LIN {X 0.154,Y -380.012,Z 1004.456,A 0.000,B 0.000,C 90.000,E1 82.129} C_DIS
LIN {X 0.169,Y -370.321,Z 1004.447,A 0.000,B 0.000,C 90.000,E1 80.387} C_DIS
LIN {X 0.082,Y -360.354,Z 1004.437,A 0.000,B 0.000,C 90.000,E1 78.634} C_DIS
LIN {X 0.041,Y -345.465,Z 1004.422,A 0.000,B 0.000,C 90.000,E1 75.936} C_DIS
LIN {X -0.138,Y -331.066,Z 1004.406,A 0.000,B 0.000,C 90.000,E1 73.196} C_DIS
LIN {X -0.138,Y -318.755,Z 1004.393,A 0.000,B 0.000,C 90.000,E1 70.678} C_DIS
LIN {X -0.044,Y -308.159,Z 1004.380,A 0.000,B 0.000,C 90.000,E1 68.411} C_DIS
LIN {X -0.184,Y -294.870,Z 1004.364,A 0.000,B 0.000,C 90.000,E1 65.485} C_DIS
LIN {X -0.128,Y -284.811,Z 1004.351,A 0.000,B 0.000,C 90.000,E1 63.127} C_DIS
LIN {X -0.028,Y -274.834,Z 1004.337,A 0.000,B 0.000,C 90.000,E1 60.717} C_DIS
LIN {X -0.023,Y -264.962,Z 1004.324,A 0.000,B 0.000,C 90.000,E1 58.280} C_DIS
LIN {X 0.089,Y -252.725,Z 1004.306,A 0.000,B 0.000,C 90.000,E1 55.055} C_DIS
LIN {X -0.103,Y -242.379,Z 1004.290,A 0.000,B 0.000,C 90.000,E1 52.190} C_DIS
LIN {X -0.123,Y -231.354,Z 1004.271,A 0.000,B 0.000,C 90.000,E1 48.852} C_DIS
LIN {X -0.097,Y -222.061,Z 1004.254,A 0.000,B 0.000,C 90.000,E1 45.810} C_DIS
LIN {X 0.061,Y -212.191,Z 1004.235,A 0.000,B 0.000,C 90.000,E1 42.285} C_DIS
LIN {X 0.119,Y -203.993,Z 1004.217,A 0.000,B 0.000,C 90.000,E1 39.116} C_DIS
LIN {X 0.034,Y -196.376,Z 1004.200,A 0.000,B 0.000,C 90.000,E1 35.931} C_DIS
LIN {X 0.017,Y -189.584,Z 1004.182,A 0.000,B 0.000,C 90.000,E1 32.673} C_DIS
LIN {X 0.019,Y -183.573,Z 1004.163,A 0.000,B 0.000,C 90.000,E1 29.361} C_DIS
LIN {X -0.052,Y -178.371,Z 1004.145,A 0.000,B 0.000,C 90.000,E1 26.027} C_DIS
LIN {X -0.084,Y -173.934,Z 1004.126,A 0.000,B 0.000,C 90.000,E1 22.642} C_DIS
LIN {X -0.091,Y -170.157,Z 1004.107,A 0.000,B 0.000,C 90.000,E1 19.214} C_DIS
LIN {X 0.076,Y -166.471,Z 1004.083,A 0.000,B 0.000,C 90.000,E1 14.828} C_DIS
LIN {X -0.002,Y -163.812,Z 1004.058,A 0.000,B 0.000,C 90.000,E1 10.489} C_DIS
LIN {X 0.043,Y -161.757,Z 1004.019,A 0.000,B 0.000,C 90.000,E1 3.440} C_DIS
LIN {X 0.074,Y -163.118,Z 1003.963,A 0.000,B 0.000,C 90.000,E1 353.337} C_DIS
LIN {X -0.025,Y -165.817,Z 1003.934,A 0.000,B 0.000,C 90.000,E1 348.105} C_DIS
LIN {X -0.007,Y -169.285,Z 1003.910,A 0.000,B 0.000,C 90.000,E1 343.740} C_DIS
LIN {X -0.058,Y -172.872,Z 1003.890,A 0.000,B 0.000,C 90.000,E1 340.296} C_DIS
LIN {X -0.003,Y -177.301,Z 1003.871,A 0.000,B 0.000,C 90.000,E1 336.847} C_DIS
LIN {X -0.031,Y -182.552,Z 1003.852,A 0.000,B 0.000,C 90.000,E1 333.461} C_DIS
LIN {X 0.066,Y -188.584,Z 1003.834,A 0.000,B 0.000,C 90.000,E1 330.078} C_DIS
LIN {X 0.013,Y -195.305,Z 1003.815,A 0.000,B 0.000,C 90.000,E1 326.786} C_DIS
LIN {X -0.035,Y -202.588,Z 1003.797,A 0.000,B 0.000,C 90.000,E1 323.543} C_DIS
LIN {X 0.095,Y -211.472,Z 1003.777,A 0.000,B 0.000,C 90.000,E1 319.908} C_DIS
LIN {X 0.122,Y -220.912,Z 1003.758,A 0.000,B 0.000,C 90.000,E1 316.377} C_DIS
LIN {X 0.094,Y -231.213,Z 1003.739,A 0.000,B 0.000,C 90.000,E1 312.933} C_DIS
LIN {X 0.048,Y -236.546,Z 1003.730,A 0.000,B 0.000,C 90.000,E1 311.434} C_DIS
LIN {X 0.068,Y -244.132,Z 1003.720,A 0.000,B 0.000,C 90.000,E1 309.564} C_DIS
LIN {X 0.061,Y -252.554,Z 1003.710,A 0.000,B 0.000,C 90.000,E1 307.729} C_DIS
LIN {X -0.082,Y -263.737,Z 1003.698,A 0.000,B 0.000,C 90.000,E1 305.598} C_DIS
LIN {X 0.083,Y -280.210,Z 1003.682,A 0.000,B 0.000,C 90.000,E1 302.752} C_DIS
LIN {X -0.015,Y -295.611,Z 1003.669,A 0.000,B 0.000,C 90.000,E1 300.384} C_DIS
LIN {X 0.092,Y -314.496,Z 1003.654,A 0.000,B 0.000,C 90.000,E1 297.719} C_DIS
LIN {X -0.130,Y -330.163,Z 1003.643,A 0.000,B 0.000,C 90.000,E1 295.848} C_DIS
LIN {X 0.087,Y -352.097,Z 1003.630,A 0.000,B 0.000,C 90.000,E1 293.462} C_DIS
LIN {X -0.028,Y -374.171,Z 1003.619,A 0.000,B 0.000,C 90.000,E1 291.354} C_DIS
LIN {X -0.007,Y -390.076,Z 1003.610,A 0.000,B 0.000,C 90.000,E1 289.885} C_DIS
LIN {X -0.151,Y -400.861,Z 1003.605,A 0.000,B 0.000,C 90.000,E1 288.906} C_DIS
LIN {X 0.103,Y -411.395,Z 1003.599,A 0.000,B 0.000,C 90.000,E1 287.873} C_DIS
LIN {X 0.172,Y -418.988,Z 1003.595,A 0.000,B 0.000,C 90.000,E1 287.094} C_DIS
LIN {X 0.026,Y -428.704,Z 1003.589,A 0.000,B 0.000,C 90.000,E1 286.079} C_DIS
LIN {X -0.072,Y -435.798,Z 1003.585,A 0.000,B 0.000,C 90.000,E1 285.300} C_DIS
LIN {X -0.131,Y -444.841,Z 1003.579,A 0.000,B 0.000,C 90.000,E1 284.245} C_DIS
LIN {X 0.030,Y -453.358,Z 1003.573,A 0.000,B 0.000,C 90.000,E1 283.175} C_DIS
LIN {X 0.188,Y -461.140,Z 1003.567,A 0.000,B 0.000,C 90.000,E1 282.119} C_DIS
LIN {X -0.108,Y -468.076,Z 1003.562,A 0.000,B 0.000,C 90.000,E1 281.130} C_DIS
LIN {X -0.096,Y -472.803,Z 1003.558,A 0.000,B 0.000,C 90.000,E1 280.366} C_DIS
LIN {X -0.133,Y -476.901,Z 1003.553,A 0.000,B 0.000,C 90.000,E1 279.613} C_DIS
LIN {X -0.128,Y -480.362,Z 1003.549,A 0.000,B 0.000,C 90.000,E1 278.859} C_DIS
LIN {X -0.094,Y -483.236,Z 1003.545,A 0.000,B 0.000,C 90.000,E1 278.106} C_DIS
LIN {X 0.077,Y -484.811,Z 1003.542,A 0.000,B 0.000,C 90.000,E1 277.587} C_DIS
LIN {X -0.222,Y -486.171,Z 1003.539,A 0.000,B 0.000,C 90.000,E1 277.125} C_DIS
LIN {X 0.173,Y -488.167,Z 1003.534,A 0.000,B 0.000,C 90.000,E1 276.087} C_DIS
LIN {X -0.104,Y -488.752,Z 1003.531,A 0.000,B 0.000,C 90.000,E1 275.625} C_DIS
LIN {X 0.108,Y -489.034,Z 1003.528,A 0.000,B 0.000,C 90.000,E1 275.106} C_DIS
LIN {X -0.166,Y -488.846,Z 1003.526,A 0.000,B 0.000,C 90.000,E1 274.645} C_DIS
LIN {X 0.012,Y -488.231,Z 1003.523,A 0.000,B 0.000,C 90.000,E1 274.131} C_DIS
LIN {X 0.224,Y -487.021,Z 1003.520,A 0.000,B 0.000,C 90.000,E1 273.612} C_DIS
LIN {X -0.084,Y -485.248,Z 1003.517,A 0.000,B 0.000,C 90.000,E1 273.154} C_DIS
LIN {X 0.113,Y -482.887,Z 1003.515,A 0.000,B 0.000,C 90.000,E1 272.636} C_DIS
LIN {X -0.211,Y -479.755,Z 1003.512,A 0.000,B 0.000,C 90.000,E1 272.178} C_DIS
LIN {X -0.054,Y -475.746,Z 1003.509,A 0.000,B 0.000,C 90.000,E1 271.661} C_DIS
LIN {X 0.065,Y -470.779,Z 1003.506,A 0.000,B 0.000,C 90.000,E1 271.146} C_DIS
LIN {X -0.119,Y -464.970,Z 1003.504,A 0.000,B 0.000,C 90.000,E1 270.688} C_DIS
LIN {X 0.155,Y -458.759,Z 1003.501,A 0.000,B 0.000,C 90.000,E1 270.229} C_DIS
LIN {X -0.051,Y -451.942,Z 1003.499,A 0.000,B 0.000,C 90.000,E1 269.885} C_DIS
LIN {X -0.182,Y -444.964,Z 1003.498,A 0.000,B 0.000,C 90.000,E1 269.599} C_DIS
LIN {X 0.077,Y -437.435,Z 1003.496,A 0.000,B 0.000,C 90.000,E1 269.312} C_DIS
LIN {X -0.119,Y -429.221,Z 1003.495,A 0.000,B 0.000,C 90.000,E1 269.141} C_DIS
LIN {X 0.095,Y -420.520,Z 1003.494,A 0.000,B 0.000,C 90.000,E1 268.969} C_DIS
LIN {X -0.086,Y -406.679,Z 1003.494,A 0.000,B 0.000,C 90.000,E1 268.854} C_DIS
LIN {X 0.121,Y -400.216,Z 1003.493,A 0.000,B 0.000,C 90.000,E1 268.797} C_DIS
LIN {X 0.026,Y -181.275,Z 1003.493,A 0.000,B 0.000,C 90.000,E1 268.797} C_DIS
LIN {X 0.089,Y -180.880,Z 1003.473,A 0.000,B 0.000,C 90.000,E1 265.065} C_DIS
LIN {X -0.032,Y -178.999,Z 1003.445,A 0.000,B 0.000,C 90.000,E1 260.038} C_DIS
LIN {X 0.062,Y -178.594,Z 1003.440,A 0.000,B 0.000,C 90.000,E1 259.162} C_DIS
LIN {X -0.044,Y -175.646,Z 1003.412,A 0.000,B 0.000,C 90.000,E1 254.102} C_DIS
LIN {X -0.039,Y -172.365,Z 1003.388,A 0.000,B 0.000,C 90.000,E1 249.826} C_DIS
LIN {X -0.024,Y -171.154,Z 1003.378,A 0.000,B 0.000,C 90.000,E1 248.103} C_DIS
LIN {X 0.020,Y -167.455,Z 1003.354,A 0.000,B 0.000,C 90.000,E1 243.768} C_DIS
LIN {X -0.046,Y -166.852,Z 1003.349,A 0.000,B 0.000,C 90.000,E1 242.922} C_DIS
LIN {X 0.018,Y -162.836,Z 1003.325,A 0.000,B 0.000,C 90.000,E1 238.535} C_DIS
LIN {X -0.007,Y -161.520,Z 1003.315,A 0.000,B 0.000,C 90.000,E1 236.786} C_DIS
LIN {X 0.034,Y -157.519,Z 1003.291,A 0.000,B 0.000,C 90.000,E1 232.351} C_DIS
LIN {X -0.033,Y -155.543,Z 1003.276,A 0.000,B 0.000,C 90.000,E1 229.703} C_DIS
LIN {X 0.009,Y -151.837,Z 1003.251,A 0.000,B 0.000,C 90.000,E1 225.202} C_DIS
LIN {X -0.083,Y -150.054,Z 1003.236,A 0.000,B 0.000,C 90.000,E1 222.528} C_DIS
LIN {X 0.042,Y -146.866,Z 1003.211,A 0.000,B 0.000,C 90.000,E1 217.935} C_DIS
LIN {X -0.060,Y -145.451,Z 1003.196,A 0.000,B 0.000,C 90.000,E1 215.231} C_DIS
LIN {X 0.054,Y -142.868,Z 1003.170,A 0.000,B 0.000,C 90.000,E1 210.590} C_DIS
LIN {X -0.020,Y -141.485,Z 1003.150,A 0.000,B 0.000,C 90.000,E1 206.924} C_DIS
LIN {X -0.034,Y -139.383,Z 1003.113,A 0.000,B 0.000,C 90.000,E1 200.429} C_DIS
LIN {X -0.046,Y -138.838,Z 1003.098,A 0.000,B 0.000,C 90.000,E1 197.638} C_DIS
LIN {X 0.015,Y -138.354,Z 1003.056,A 0.000,B 0.000,C 90.000,E1 190.141} C_DIS
LIN {X 0.010,Y -139.522,Z 1003.004,A 0.000,B 0.000,C 90.000,E1 180.802} C_DIS
LIN {X -0.050,Y -141.187,Z 1002.973,A 0.000,B 0.000,C 90.000,E1 175.241} C_DIS
LIN {X 0.063,Y -142.564,Z 1002.958,A 0.000,B 0.000,C 90.000,E1 172.413} C_DIS
LIN {X 0.018,Y -144.848,Z 1002.932,A 0.000,B 0.000,C 90.000,E1 167.813} C_DIS
LIN {X -0.027,Y -147.473,Z 1002.912,A 0.000,B 0.000,C 90.000,E1 164.157} C_DIS
LIN {X -0.001,Y -150.058,Z 1002.892,A 0.000,B 0.000,C 90.000,E1 160.496} C_DIS
LIN {X 0.004,Y -153.403,Z 1002.872,A 0.000,B 0.000,C 90.000,E1 156.869} C_DIS
LIN {X 0.051,Y -155.934,Z 1002.857,A 0.000,B 0.000,C 90.000,E1 154.152} C_DIS
LIN {X 0.024,Y -159.802,Z 1002.837,A 0.000,B 0.000,C 90.000,E1 150.589} C_DIS
LIN {X 0.010,Y -162.042,Z 1002.827,A 0.000,B 0.000,C 90.000,E1 148.820} C_DIS
LIN {X -0.016,Y -166.238,Z 1002.807,A 0.000,B 0.000,C 90.000,E1 145.308} C_DIS
LIN {X -0.015,Y -171.255,Z 1002.788,A 0.000,B 0.000,C 90.000,E1 141.823} C_DIS
LIN {X -0.093,Y -176.144,Z 1002.769,A 0.000,B 0.000,C 90.000,E1 138.405} C_DIS
LIN {X 0.023,Y -180.413,Z 1002.755,A 0.000,B 0.000,C 90.000,E1 135.810} C_DIS
LIN {X -0.001,Y -185.819,Z 1002.736,A 0.000,B 0.000,C 90.000,E1 132.447} C_DIS
LIN {X 0.053,Y -190.439,Z 1002.722,A 0.000,B 0.000,C 90.000,E1 129.930} C_DIS
LIN {X -0.111,Y -196.231,Z 1002.703,A 0.000,B 0.000,C 90.000,E1 126.664} C_DIS
LIN {X -0.025,Y -300.780,Z 1002.703,A 0.000,B 0.000,C 90.000,E1 126.629} C_DIS
LIN {X 0.004,Y -302.851,Z 1002.703,A 0.000,B 0.000,C 90.000,E1 126.583} C_DIS
LIN {X 0.105,Y -306.723,Z 1002.702,A 0.000,B 0.000,C 90.000,E1 126.377} C_DIS
LIN {X -0.041,Y -309.025,Z 1002.701,A 0.000,B 0.000,C 90.000,E1 126.217} C_DIS
LIN {X 0.165,Y -312.203,Z 1002.699,A 0.000,B 0.000,C 90.000,E1 125.804} C_DIS
LIN {X -0.006,Y -314.146,Z 1002.697,A 0.000,B 0.000,C 90.000,E1 125.518} C_DIS
LIN {X 0.080,Y -315.663,Z 1002.696,A 0.000,B 0.000,C 90.000,E1 125.185} C_DIS
LIN {X 0.120,Y -317.903,Z 1002.692,A 0.000,B 0.000,C 90.000,E1 124.532} C_DIS
LIN {X -0.113,Y -328.902,Z 1002.674,A 0.000,B 0.000,C 90.000,E1 121.386} C_DIS
LIN {X -0.080,Y -340.185,Z 1002.659,A 0.000,B 0.000,C 90.000,E1 118.565} C_DIS
LIN {X -0.035,Y -352.884,Z 1002.643,A 0.000,B 0.000,C 90.000,E1 115.796} C_DIS
LIN {X 0.074,Y -367.106,Z 1002.628,A 0.000,B 0.000,C 90.000,E1 113.078} C_DIS
LIN {X 0.030,Y -381.133,Z 1002.615,A 0.000,B 0.000,C 90.000,E1 110.737} C_DIS
LIN {X 0.205,Y -396.566,Z 1002.602,A 0.000,B 0.000,C 90.000,E1 108.417} C_DIS
LIN {X 0.011,Y -413.514,Z 1002.590,A 0.000,B 0.000,C 90.000,E1 106.205} C_DIS
LIN {X 0.123,Y -432.099,Z 1002.578,A 0.000,B 0.000,C 90.000,E1 104.008} C_DIS
LIN {X -0.022,Y -451.998,Z 1002.566,A 0.000,B 0.000,C 90.000,E1 101.951} C_DIS
LIN {X 0.102,Y -467.286,Z 1002.558,A 0.000,B 0.000,C 90.000,E1 100.489} C_DIS
LIN {X 0.122,Y -469.335,Z 1002.557,A 0.000,B 0.000,C 90.000,E1 100.254} C_DIS
LIN {X -0.030,Y -471.015,Z 1002.556,A 0.000,B 0.000,C 90.000,E1 100.018} C_DIS
LIN {X -0.183,Y -472.276,Z 1002.554,A 0.000,B 0.000,C 90.000,E1 99.782} C_DIS
LIN {X -0.082,Y -473.833,Z 1002.551,A 0.000,B 0.000,C 90.000,E1 99.265} C_DIS
LIN {X 0.030,Y -474.341,Z 1002.549,A 0.000,B 0.000,C 90.000,E1 98.746} C_DIS
LIN {X 0.223,Y -473.887,Z 1002.546,A 0.000,B 0.000,C 90.000,E1 98.219} C_DIS
LIN {X -0.121,Y -472.404,Z 1002.543,A 0.000,B 0.000,C 90.000,E1 97.757} C_DIS
LIN {X 0.145,Y -471.200,Z 1002.542,A 0.000,B 0.000,C 90.000,E1 97.473} C_DIS
LIN {X 0.112,Y -466.100,Z 1002.537,A 0.000,B 0.000,C 90.000,E1 96.720} C_DIS
LIN {X -0.140,Y -455.701,Z 1002.529,A 0.000,B 0.000,C 90.000,E1 95.220} C_DIS
LIN {X -0.105,Y -436.571,Z 1002.513,A 0.000,B 0.000,C 90.000,E1 92.350} C_DIS
LIN {X 0.100,Y -425.250,Z 1002.503,A 0.000,B 0.000,C 90.000,E1 90.458} C_DIS
LIN {X 0.013,Y -408.885,Z 1002.486,A 0.000,B 0.000,C 90.000,E1 87.478} C_DIS
LIN {X 0.033,Y -399.955,Z 1002.477,A 0.000,B 0.000,C 90.000,E1 85.812} C_DIS
LIN {X -0.051,Y -389.282,Z 1002.466,A 0.000,B 0.000,C 90.000,E1 83.856} C_DIS
LIN {X 0.037,Y -379.912,Z 1002.456,A 0.000,B 0.000,C 90.000,E1 82.129} C_DIS
LIN {X 0.054,Y -370.238,Z 1002.447,A 0.000,B 0.000,C 90.000,E1 80.387} C_DIS
LIN {X -0.032,Y -360.282,Z 1002.437,A 0.000,B 0.000,C 90.000,E1 78.634} C_DIS
LIN {X -0.070,Y -345.356,Z 1002.422,A 0.000,B 0.000,C 90.000,E1 75.936} C_DIS
LIN {X 0.068,Y -330.961,Z 1002.406,A 0.000,B 0.000,C 90.000,E1 73.142} C_DIS
LIN {X 0.160,Y -318.687,Z 1002.392,A 0.000,B 0.000,C 90.000,E1 70.604} C_DIS
LIN {X -0.151,Y -308.077,Z 1002.380,A 0.000,B 0.000,C 90.000,E1 68.411} C_DIS
LIN {X 0.104,Y -294.795,Z 1002.364,A 0.000,B 0.000,C 90.000,E1 65.409} C_DIS
LIN {X 0.025,Y -284.744,Z 1002.350,A 0.000,B 0.000,C 90.000,E1 63.076} C_DIS
LIN {X 0.112,Y -274.750,Z 1002.337,A 0.000,B 0.000,C 90.000,E1 60.667} C_DIS
LIN {X -0.061,Y -263.473,Z 1002.322,A 0.000,B 0.000,C 90.000,E1 57.916} C_DIS
LIN {X 0.016,Y -251.296,Z 1002.304,A 0.000,B 0.000,C 90.000,E1 54.689} C_DIS
LIN {X -0.020,Y -239.775,Z 1002.286,A 0.000,B 0.000,C 90.000,E1 51.412} C_DIS
LIN {X 0.025,Y -228.872,Z 1002.267,A 0.000,B 0.000,C 90.000,E1 48.038} C_DIS
LIN {X 0.050,Y -218.580,Z 1002.248,A 0.000,B 0.000,C 90.000,E1 44.595} C_DIS
LIN {X -0.069,Y -209.973,Z 1002.231,A 0.000,B 0.000,C 90.000,E1 41.515} C_DIS
LIN {X -0.033,Y -201.928,Z 1002.213,A 0.000,B 0.000,C 90.000,E1 38.338} C_DIS
LIN {X 0.002,Y -194.542,Z 1002.195,A 0.000,B 0.000,C 90.000,E1 35.105} C_DIS
LIN {X 0.101,Y -187.950,Z 1002.177,A 0.000,B 0.000,C 90.000,E1 31.799} C_DIS
LIN {X 0.061,Y -182.166,Z 1002.158,A 0.000,B 0.000,C 90.000,E1 28.487} C_DIS
LIN {X -0.051,Y -177.168,Z 1002.140,A 0.000,B 0.000,C 90.000,E1 25.155} C_DIS
LIN {X 0.053,Y -172.900,Z 1002.121,A 0.000,B 0.000,C 90.000,E1 21.716} C_DIS
LIN {X -0.039,Y -169.318,Z 1002.102,A 0.000,B 0.000,C 90.000,E1 18.308} C_DIS
LIN {X 0.013,Y -165.847,Z 1002.078,A 0.000,B 0.000,C 90.000,E1 13.953} C_DIS
LIN {X 0.054,Y -163.078,Z 1002.048,A 0.000,B 0.000,C 90.000,E1 8.690} C_DIS
LIN {X 0.006,Y -163.856,Z 1001.953,A 0.000,B 0.000,C 90.000,E1 351.602} C_DIS
LIN {X -0.017,Y -166.435,Z 1001.929,A 0.000,B 0.000,C 90.000,E1 347.229} C_DIS
LIN {X 0.057,Y -170.137,Z 1001.905,A 0.000,B 0.000,C 90.000,E1 342.851} C_DIS
LIN {X 0.079,Y -173.939,Z 1001.886,A 0.000,B 0.000,C 90.000,E1 339.390} C_DIS
LIN {X -0.009,Y -178.575,Z 1001.867,A 0.000,B 0.000,C 90.000,E1 335.997} C_DIS
LIN {X -0.018,Y -184.040,Z 1001.848,A 0.000,B 0.000,C 90.000,E1 332.615} C_DIS
LIN {X -0.047,Y -190.271,Z 1001.829,A 0.000,B 0.000,C 90.000,E1 329.282} C_DIS
LIN {X 0.044,Y -197.117,Z 1001.811,A 0.000,B 0.000,C 90.000,E1 325.960} C_DIS
LIN {X 0.041,Y -204.566,Z 1001.793,A 0.000,B 0.000,C 90.000,E1 322.718} C_DIS
LIN {X 0.032,Y -213.593,Z 1001.773,A 0.000,B 0.000,C 90.000,E1 319.138} C_DIS
LIN {X -0.043,Y -223.147,Z 1001.754,A 0.000,B 0.000,C 90.000,E1 315.648} C_DIS
LIN {X 0.101,Y -231.183,Z 1001.739,A 0.000,B 0.000,C 90.000,E1 312.933} C_DIS
LIN {X 0.055,Y -236.542,Z 1001.730,A 0.000,B 0.000,C 90.000,E1 311.434} C_DIS
LIN {X 0.066,Y -245.822,Z 1001.718,A 0.000,B 0.000,C 90.000,E1 309.197} C_DIS
LIN {X 0.081,Y -254.420,Z 1001.708,A 0.000,B 0.000,C 90.000,E1 307.363} C_DIS
LIN {X -0.125,Y -267.785,Z 1001.694,A 0.000,B 0.000,C 90.000,E1 304.898} C_DIS
LIN {X -0.006,Y -284.641,Z 1001.678,A 0.000,B 0.000,C 90.000,E1 302.084} C_DIS
LIN {X -0.140,Y -304.900,Z 1001.661,A 0.000,B 0.000,C 90.000,E1 299.077} C_DIS
LIN {X 0.075,Y -319.636,Z 1001.651,A 0.000,B 0.000,C 90.000,E1 297.078} C_DIS
LIN {X -0.039,Y -335.857,Z 1001.640,A 0.000,B 0.000,C 90.000,E1 295.207} C_DIS
LIN {X -0.083,Y -355.063,Z 1001.629,A 0.000,B 0.000,C 90.000,E1 293.206} C_DIS
LIN {X -0.172,Y -373.890,Z 1001.619,A 0.000,B 0.000,C 90.000,E1 291.408} C_DIS
LIN {X 0.029,Y -390.042,Z 1001.610,A 0.000,B 0.000,C 90.000,E1 289.885} C_DIS
LIN {X -0.120,Y -403.318,Z 1001.604,A 0.000,B 0.000,C 90.000,E1 288.671} C_DIS
LIN {X 0.193,Y -411.201,Z 1001.599,A 0.000,B 0.000,C 90.000,E1 287.873} C_DIS
LIN {X 0.238,Y -418.847,Z 1001.595,A 0.000,B 0.000,C 90.000,E1 287.094} C_DIS
LIN {X -0.109,Y -428.758,Z 1001.589,A 0.000,B 0.000,C 90.000,E1 286.079} C_DIS
LIN {X 0.123,Y -435.945,Z 1001.585,A 0.000,B 0.000,C 90.000,E1 285.245} C_DIS
LIN {X 0.073,Y -444.940,Z 1001.579,A 0.000,B 0.000,C 90.000,E1 284.189} C_DIS
LIN {X 0.240,Y -453.474,Z 1001.573,A 0.000,B 0.000,C 90.000,E1 283.119} C_DIS
LIN {X 0.133,Y -459.356,Z 1001.569,A 0.000,B 0.000,C 90.000,E1 282.355} C_DIS
LIN {X -0.184,Y -466.509,Z 1001.563,A 0.000,B 0.000,C 90.000,E1 281.366} C_DIS
LIN {X -0.189,Y -471.390,Z 1001.559,A 0.000,B 0.000,C 90.000,E1 280.602} C_DIS
LIN {X -0.234,Y -475.696,Z 1001.555,A 0.000,B 0.000,C 90.000,E1 279.849} C_DIS
LIN {X -0.167,Y -479.383,Z 1001.550,A 0.000,B 0.000,C 90.000,E1 279.086} C_DIS
LIN {X -0.020,Y -481.514,Z 1001.548,A 0.000,B 0.000,C 90.000,E1 278.568} C_DIS
LIN {X 0.144,Y -483.361,Z 1001.545,A 0.000,B 0.000,C 90.000,E1 278.049} C_DIS
LIN {X -0.164,Y -484.952,Z 1001.542,A 0.000,B 0.000,C 90.000,E1 277.587} C_DIS
LIN {X 0.020,Y -486.323,Z 1001.539,A 0.000,B 0.000,C 90.000,E1 277.068} C_DIS
LIN {X 0.215,Y -487.451,Z 1001.536,A 0.000,B 0.000,C 90.000,E1 276.549} C_DIS
LIN {X -0.067,Y -488.308,Z 1001.534,A 0.000,B 0.000,C 90.000,E1 276.087} C_DIS
LIN {X 0.143,Y -488.899,Z 1001.531,A 0.000,B 0.000,C 90.000,E1 275.568} C_DIS
LIN {X -0.131,Y -489.104,Z 1001.528,A 0.000,B 0.000,C 90.000,E1 275.106} C_DIS
LIN {X 0.084,Y -488.932,Z 1001.526,A 0.000,B 0.000,C 90.000,E1 274.588} C_DIS
LIN {X -0.225,Y -488.308,Z 1001.523,A 0.000,B 0.000,C 90.000,E1 274.131} C_DIS
LIN {X -0.012,Y -487.129,Z 1001.520,A 0.000,B 0.000,C 90.000,E1 273.612} C_DIS
LIN {X 0.193,Y -485.347,Z 1001.517,A 0.000,B 0.000,C 90.000,E1 273.094} C_DIS
LIN {X -0.120,Y -482.933,Z 1001.515,A 0.000,B 0.000,C 90.000,E1 272.636} C_DIS
LIN {X 0.038,Y -479.770,Z 1001.512,A 0.000,B 0.000,C 90.000,E1 272.121} C_DIS
LIN {X 0.193,Y -475.730,Z 1001.509,A 0.000,B 0.000,C 90.000,E1 271.604} C_DIS
LIN {X -0.161,Y -470.689,Z 1001.506,A 0.000,B 0.000,C 90.000,E1 271.146} C_DIS
LIN {X -0.233,Y -467.980,Z 1001.505,A 0.000,B 0.000,C 90.000,E1 270.917} C_DIS
LIN {X -0.157,Y -461.996,Z 1001.502,A 0.000,B 0.000,C 90.000,E1 270.458} C_DIS
LIN {X -0.087,Y -455.556,Z 1001.500,A 0.000,B 0.000,C 90.000,E1 270.057} C_DIS
LIN {X 0.006,Y -448.671,Z 1001.498,A 0.000,B 0.000,C 90.000,E1 269.714} C_DIS
LIN {X 0.090,Y -441.537,Z 1001.497,A 0.000,B 0.000,C 90.000,E1 269.427} C_DIS
LIN {X 0.141,Y -433.909,Z 1001.496,A 0.000,B 0.000,C 90.000,E1 269.198} C_DIS
LIN {X 0.159,Y -425.715,Z 1001.495,A 0.000,B 0.000,C 90.000,E1 269.026} C_DIS
LIN {X 0.096,Y -417.151,Z 1001.494,A 0.000,B 0.000,C 90.000,E1 268.912} C_DIS
LIN {X 0.117,Y -404.897,Z 1001.493,A 0.000,B 0.000,C 90.000,E1 268.797} C_DIS
LIN {X -0.025,Y -399.475,Z 1001.493,A 0.000,B 0.000,C 90.000,E1 268.797} C_DIS
LIN {X -0.032,Y -181.272,Z 1001.493,A 0.000,B 0.000,C 90.000,E1 268.797} C_DIS
LIN {X 0.048,Y -180.906,Z 1001.474,A 0.000,B 0.000,C 90.000,E1 265.355} C_DIS
LIN {X -0.059,Y -180.690,Z 1001.470,A 0.000,B 0.000,C 90.000,E1 264.546} C_DIS
LIN {X 0.019,Y -178.773,Z 1001.441,A 0.000,B 0.000,C 90.000,E1 259.454} C_DIS
LIN {X -0.078,Y -175.819,Z 1001.413,A 0.000,B 0.000,C 90.000,E1 254.393} C_DIS
LIN {X -0.076,Y -172.008,Z 1001.385,A 0.000,B 0.000,C 90.000,E1 249.263} C_DIS
LIN {X -0.100,Y -171.425,Z 1001.380,A 0.000,B 0.000,C 90.000,E1 248.411} C_DIS
LIN {X -0.044,Y -167.663,Z 1001.356,A 0.000,B 0.000,C 90.000,E1 244.076} C_DIS
LIN {X -0.104,Y -166.333,Z 1001.346,A 0.000,B 0.000,C 90.000,E1 242.359} C_DIS
LIN {X 0.029,Y -163.070,Z 1001.327,A 0.000,B 0.000,C 90.000,E1 238.820} C_DIS
LIN {X -0.059,Y -161.009,Z 1001.312,A 0.000,B 0.000,C 90.000,E1 236.215} C_DIS
LIN {X 0.051,Y -157.753,Z 1001.293,A 0.000,B 0.000,C 90.000,E1 232.637} C_DIS
LIN {X -0.011,Y -155.791,Z 1001.278,A 0.000,B 0.000,C 90.000,E1 229.989} C_DIS
LIN {X 0.044,Y -152.044,Z 1001.253,A 0.000,B 0.000,C 90.000,E1 225.486} C_DIS
LIN {X 0.062,Y -150.294,Z 1001.238,A 0.000,B 0.000,C 90.000,E1 222.771} C_DIS
LIN {X -0.013,Y -147.041,Z 1001.213,A 0.000,B 0.000,C 90.000,E1 218.257} C_DIS
LIN {X -0.021,Y -145.621,Z 1001.197,A 0.000,B 0.000,C 90.000,E1 215.518} C_DIS
LIN {X -0.021,Y -143.005,Z 1001.172,A 0.000,B 0.000,C 90.000,E1 210.924} C_DIS
LIN {X 0.036,Y -141.631,Z 1001.151,A 0.000,B 0.000,C 90.000,E1 207.206} C_DIS
LIN {X -0.039,Y -139.436,Z 1001.115,A 0.000,B 0.000,C 90.000,E1 200.737} C_DIS
LIN {X 0.015,Y -139.167,Z 1001.105,A 0.000,B 0.000,C 90.000,E1 198.852} C_DIS
LIN {X 0.048,Y -138.317,Z 1001.053,A 0.000,B 0.000,C 90.000,E1 189.500} C_DIS
LIN {X 0.059,Y -139.475,Z 1001.006,A 0.000,B 0.000,C 90.000,E1 181.088} C_DIS
LIN {X 0.001,Y -141.055,Z 1000.975,A 0.000,B 0.000,C 90.000,E1 175.527} C_DIS
LIN {X -0.045,Y -142.427,Z 1000.960,A 0.000,B 0.000,C 90.000,E1 172.761} C_DIS
LIN {X 0.016,Y -144.664,Z 1000.934,A 0.000,B 0.000,C 90.000,E1 168.117} C_DIS
LIN {X -0.001,Y -147.247,Z 1000.914,A 0.000,B 0.000,C 90.000,E1 164.448} C_DIS
LIN {X 0.017,Y -150.565,Z 1000.888,A 0.000,B 0.000,C 90.000,E1 159.880} C_DIS
LIN {X -0.044,Y -154.033,Z 1000.868,A 0.000,B 0.000,C 90.000,E1 156.282} C_DIS
LIN {X 0.024,Y -157.449,Z 1000.848,A 0.000,B 0.000,C 90.000,E1 152.666} C_DIS
LIN {X -0.027,Y -161.667,Z 1000.828,A 0.000,B 0.000,C 90.000,E1 149.125} C_DIS
LIN {X -0.010,Y -165.862,Z 1000.809,A 0.000,B 0.000,C 90.000,E1 145.595} C_DIS
LIN {X -0.019,Y -170.839,Z 1000.789,A 0.000,B 0.000,C 90.000,E1 142.110} C_DIS
LIN {X 0.029,Y -175.708,Z 1000.770,A 0.000,B 0.000,C 90.000,E1 138.647} C_DIS
LIN {X 0.020,Y -181.319,Z 1000.751,A 0.000,B 0.000,C 90.000,E1 135.243} C_DIS
LIN {X -0.109,Y -186.804,Z 1000.733,A 0.000,B 0.000,C 90.000,E1 131.919} C_DIS
LIN {X -0.039,Y -191.395,Z 1000.719,A 0.000,B 0.000,C 90.000,E1 129.402} C_DIS
LIN {X 0.039,Y -196.149,Z 1000.704,A 0.000,B 0.000,C 90.000,E1 126.664} C_DIS
LIN {X 0.012,Y -300.415,Z 1000.704,A 0.000,B 0.000,C 90.000,E1 126.664} C_DIS
LIN {X -0.037,Y -301.224,Z 1000.704,A 0.000,B 0.000,C 90.000,E1 126.664} C_DIS
LIN {X 0.015,Y -307.356,Z 1000.702,A 0.000,B 0.000,C 90.000,E1 126.377} C_DIS
LIN {X 0.068,Y -310.274,Z 1000.701,A 0.000,B 0.000,C 90.000,E1 126.091} C_DIS
LIN {X -0.190,Y -313.967,Z 1000.698,A 0.000,B 0.000,C 90.000,E1 125.598} C_DIS
LIN {X 0.037,Y -315.520,Z 1000.696,A 0.000,B 0.000,C 90.000,E1 125.231} C_DIS
LIN {X -0.113,Y -317.762,Z 1000.692,A 0.000,B 0.000,C 90.000,E1 124.612} C_DIS
LIN {X 0.098,Y -328.744,Z 1000.674,A 0.000,B 0.000,C 90.000,E1 121.386} C_DIS
LIN {X 0.130,Y -340.011,Z 1000.659,A 0.000,B 0.000,C 90.000,E1 118.565} C_DIS
LIN {X -0.135,Y -352.688,Z 1000.643,A 0.000,B 0.000,C 90.000,E1 115.848} C_DIS
LIN {X -0.049,Y -366.894,Z 1000.628,A 0.000,B 0.000,C 90.000,E1 113.131} C_DIS
LIN {X -0.108,Y -380.902,Z 1000.615,A 0.000,B 0.000,C 90.000,E1 110.791} C_DIS
LIN {X -0.076,Y -396.314,Z 1000.603,A 0.000,B 0.000,C 90.000,E1 108.489} C_DIS
LIN {X -0.163,Y -413.240,Z 1000.590,A 0.000,B 0.000,C 90.000,E1 106.260} C_DIS
LIN {X -0.070,Y -431.801,Z 1000.578,A 0.000,B 0.000,C 90.000,E1 104.064} C_DIS
LIN {X 0.184,Y -451.703,Z 1000.567,A 0.000,B 0.000,C 90.000,E1 101.951} C_DIS
LIN {X -0.158,Y -467.004,Z 1000.558,A 0.000,B 0.000,C 90.000,E1 100.546} C_DIS
LIN {X -0.152,Y -469.136,Z 1000.557,A 0.000,B 0.000,C 90.000,E1 100.310} C_DIS
LIN {X -0.149,Y -470.750,Z 1000.556,A 0.000,B 0.000,C 90.000,E1 100.074} C_DIS
LIN {X 0.088,Y -472.073,Z 1000.554,A 0.000,B 0.000,C 90.000,E1 99.792} C_DIS
LIN {X -0.059,Y -473.051,Z 1000.553,A 0.000,B 0.000,C 90.000,E1 99.557} C_DIS
LIN {X 0.126,Y -474.153,Z 1000.550,A 0.000,B 0.000,C 90.000,E1 99.029} C_DIS
LIN {X -0.227,Y -474.265,Z 1000.547,A 0.000,B 0.000,C 90.000,E1 98.568} C_DIS
LIN {X -0.101,Y -473.404,Z 1000.545,A 0.000,B 0.000,C 90.000,E1 98.049} C_DIS
LIN {X 0.025,Y -471.432,Z 1000.542,A 0.000,B 0.000,C 90.000,E1 97.530} C_DIS
LIN {X 0.148,Y -468.162,Z 1000.539,A 0.000,B 0.000,C 90.000,E1 97.011} C_DIS
LIN {X 0.203,Y -456.059,Z 1000.529,A 0.000,B 0.000,C 90.000,E1 95.220} C_DIS
LIN {X -0.198,Y -436.892,Z 1000.513,A 0.000,B 0.000,C 90.000,E1 92.407} C_DIS
LIN {X 0.145,Y -424.016,Z 1000.501,A 0.000,B 0.000,C 90.000,E1 90.229} C_DIS
LIN {X -0.059,Y -409.188,Z 1000.486,A 0.000,B 0.000,C 90.000,E1 87.535} C_DIS
LIN {X -0.030,Y -400.253,Z 1000.477,A 0.000,B 0.000,C 90.000,E1 85.869} C_DIS
LIN {X -0.162,Y -391.113,Z 1000.468,A 0.000,B 0.000,C 90.000,E1 84.204} C_DIS
LIN {X 0.011,Y -381.785,Z 1000.458,A 0.000,B 0.000,C 90.000,E1 82.470} C_DIS
LIN {X 0.011,Y -372.157,Z 1000.449,A 0.000,B 0.000,C 90.000,E1 80.735} C_DIS
LIN {X -0.090,Y -363.950,Z 1000.440,A 0.000,B 0.000,C 90.000,E1 79.285} C_DIS
LIN {X 0.027,Y -350.582,Z 1000.427,A 0.000,B 0.000,C 90.000,E1 76.881} C_DIS
LIN {X -0.110,Y -335.979,Z 1000.412,A 0.000,B 0.000,C 90.000,E1 74.157} C_DIS
LIN {X -0.037,Y -322.015,Z 1000.396,A 0.000,B 0.000,C 90.000,E1 71.329} C_DIS
LIN {X 0.027,Y -311.402,Z 1000.384,A 0.000,B 0.000,C 90.000,E1 69.082} C_DIS
LIN {X -0.147,Y -297.987,Z 1000.367,A 0.000,B 0.000,C 90.000,E1 66.177} C_DIS
LIN {X 0.088,Y -286.424,Z 1000.353,A 0.000,B 0.000,C 90.000,E1 63.461} C_DIS
LIN {X -0.031,Y -276.429,Z 1000.339,A 0.000,B 0.000,C 90.000,E1 61.101} C_DIS
LIN {X -0.062,Y -265.075,Z 1000.324,A 0.000,B 0.000,C 90.000,E1 58.329} C_DIS
LIN {X 0.059,Y -252.819,Z 1000.306,A 0.000,B 0.000,C 90.000,E1 55.102} C_DIS
LIN {X 0.067,Y -241.201,Z 1000.288,A 0.000,B 0.000,C 90.000,E1 51.823} C_DIS
LIN {X 0.005,Y -230.195,Z 1000.269,A 0.000,B 0.000,C 90.000,E1 48.485} C_DIS
LIN {X -0.008,Y -220.932,Z 1000.252,A 0.000,B 0.000,C 90.000,E1 45.445} C_DIS
LIN {X -0.030,Y -211.149,Z 1000.233,A 0.000,B 0.000,C 90.000,E1 41.962} C_DIS
LIN {X -0.128,Y -203.034,Z 1000.216,A 0.000,B 0.000,C 90.000,E1 38.830} C_DIS
LIN {X -0.065,Y -195.561,Z 1000.198,A 0.000,B 0.000,C 90.000,E1 35.598} C_DIS
LIN {X -0.095,Y -188.857,Z 1000.180,A 0.000,B 0.000,C 90.000,E1 32.339} C_DIS
LIN {X -0.017,Y -182.969,Z 1000.161,A 0.000,B 0.000,C 90.000,E1 28.999} C_DIS
LIN {X -0.032,Y -177.852,Z 1000.142,A 0.000,B 0.000,C 90.000,E1 25.643} C_DIS
LIN {X 0.082,Y -173.500,Z 1000.124,A 0.000,B 0.000,C 90.000,E1 22.206} C_DIS
LIN {X 0.057,Y -169.790,Z 1000.104,A 0.000,B 0.000,C 90.000,E1 18.779} C_DIS
LIN {X -0.045,Y -166.211,Z 1000.080,A 0.000,B 0.000,C 90.000,E1 14.481} C_DIS
LIN {X 0.067,Y -163.665,Z 1000.056,A 0.000,B 0.000,C 90.000,E1 10.074} C_DIS
LIN {X 0.073,Y -161.722,Z 1000.017,A 0.000,B 0.000,C 90.000,E1 3.037} C_DIS
LIN {X 0.075,Y -163.132,Z 999.963,A 0.000,B 0.000,C 90.000,E1 353.337} C_DIS
LIN {X -0.024,Y -165.837,Z 999.934,A 0.000,B 0.000,C 90.000,E1 348.105} C_DIS
LIN {X -0.005,Y -169.337,Z 999.910,A 0.000,B 0.000,C 90.000,E1 343.740} C_DIS
LIN {X -0.055,Y -172.954,Z 999.890,A 0.000,B 0.000,C 90.000,E1 340.296} C_DIS
LIN {X 0.003,Y -177.405,Z 999.871,A 0.000,B 0.000,C 90.000,E1 336.847} C_DIS
LIN {X -0.023,Y -182.661,Z 999.853,A 0.000,B 0.000,C 90.000,E1 333.461} C_DIS
LIN {X -0.086,Y -188.710,Z 999.834,A 0.000,B 0.000,C 90.000,E1 330.127} C_DIS
LIN {X 0.028,Y -195.430,Z 999.816,A 0.000,B 0.000,C 90.000,E1 326.786} C_DIS
LIN {X -0.016,Y -202.728,Z 999.797,A 0.000,B 0.000,C 90.000,E1 323.543} C_DIS
LIN {X 0.113,Y -211.618,Z 999.777,A 0.000,B 0.000,C 90.000,E1 319.908} C_DIS
LIN {X -0.015,Y -220.999,Z 999.758,A 0.000,B 0.000,C 90.000,E1 316.419} C_DIS
LIN {X -0.050,Y -231.148,Z 999.739,A 0.000,B 0.000,C 90.000,E1 312.975} C_DIS
LIN {X 0.072,Y -236.556,Z 999.730,A 0.000,B 0.000,C 90.000,E1 311.434} C_DIS
LIN {X 0.085,Y -245.905,Z 999.718,A 0.000,B 0.000,C 90.000,E1 309.197} C_DIS
LIN {X 0.103,Y -254.512,Z 999.708,A 0.000,B 0.000,C 90.000,E1 307.363} C_DIS
LIN {X -0.100,Y -267.860,Z 999.694,A 0.000,B 0.000,C 90.000,E1 304.898} C_DIS
LIN {X 0.021,Y -284.712,Z 999.678,A 0.000,B 0.000,C 90.000,E1 302.084} C_DIS
LIN {X -0.108,Y -304.959,Z 999.661,A 0.000,B 0.000,C 90.000,E1 299.077} C_DIS
LIN {X -0.083,Y -317.098,Z 999.652,A 0.000,B 0.000,C 90.000,E1 297.436} C_DIS
LIN {X -0.066,Y -332.988,Z 999.642,A 0.000,B 0.000,C 90.000,E1 295.540} C_DIS
LIN {X 0.145,Y -354.800,Z 999.629,A 0.000,B 0.000,C 90.000,E1 293.206} C_DIS
LIN {X -0.031,Y -373.724,Z 999.619,A 0.000,B 0.000,C 90.000,E1 291.408} C_DIS
LIN {X 0.045,Y -390.036,Z 999.611,A 0.000,B 0.000,C 90.000,E1 289.885} C_DIS
LIN {X -0.112,Y -403.278,Z 999.604,A 0.000,B 0.000,C 90.000,E1 288.671} C_DIS
LIN {X 0.205,Y -411.129,Z 999.599,A 0.000,B 0.000,C 90.000,E1 287.873} C_DIS
LIN {X 0.239,Y -418.765,Z 999.595,A 0.000,B 0.000,C 90.000,E1 287.094} C_DIS
LIN {X -0.153,Y -428.703,Z 999.589,A 0.000,B 0.000,C 90.000,E1 286.079} C_DIS
LIN {X 0.056,Y -435.912,Z 999.585,A 0.000,B 0.000,C 90.000,E1 285.245} C_DIS
LIN {X -0.097,Y -447.063,Z 999.577,A 0.000,B 0.000,C 90.000,E1 283.939} C_DIS
LIN {X -0.019,Y -455.425,Z 999.572,A 0.000,B 0.000,C 90.000,E1 282.883} C_DIS
LIN {X -0.119,Y -461.157,Z 999.567,A 0.000,B 0.000,C 90.000,E1 282.119} C_DIS
LIN {X 0.040,Y -468.132,Z 999.562,A 0.000,B 0.000,C 90.000,E1 281.074} C_DIS
LIN {X 0.055,Y -472.877,Z 999.557,A 0.000,B 0.000,C 90.000,E1 280.310} C_DIS
LIN {X 0.022,Y -477.005,Z 999.553,A 0.000,B 0.000,C 90.000,E1 279.557} C_DIS
LIN {X 0.029,Y -480.513,Z 999.549,A 0.000,B 0.000,C 90.000,E1 278.803} C_DIS
LIN {X 0.066,Y -483.415,Z 999.545,A 0.000,B 0.000,C 90.000,E1 278.049} C_DIS
LIN {X -0.241,Y -485.029,Z 999.542,A 0.000,B 0.000,C 90.000,E1 277.587} C_DIS
LIN {X 0.138,Y -487.571,Z 999.536,A 0.000,B 0.000,C 90.000,E1 276.549} C_DIS
LIN {X -0.143,Y -488.419,Z 999.534,A 0.000,B 0.000,C 90.000,E1 276.087} C_DIS
LIN {X 0.067,Y -489.015,Z 999.531,A 0.000,B 0.000,C 90.000,E1 275.568} C_DIS
LIN {X -0.206,Y -489.244,Z 999.528,A 0.000,B 0.000,C 90.000,E1 275.106} C_DIS
LIN {X 0.010,Y -489.057,Z 999.526,A 0.000,B 0.000,C 90.000,E1 274.588} C_DIS
LIN {X 0.188,Y -488.423,Z 999.523,A 0.000,B 0.000,C 90.000,E1 274.073} C_DIS
LIN {X -0.085,Y -487.216,Z 999.520,A 0.000,B 0.000,C 90.000,E1 273.612} C_DIS
LIN {X 0.121,Y -485.482,Z 999.517,A 0.000,B 0.000,C 90.000,E1 273.094} C_DIS
LIN {X -0.191,Y -483.073,Z 999.515,A 0.000,B 0.000,C 90.000,E1 272.636} C_DIS
LIN {X 0.128,Y -481.600,Z 999.513,A 0.000,B 0.000,C 90.000,E1 272.350} C_DIS
LIN {X -0.200,Y -478.023,Z 999.510,A 0.000,B 0.000,C 90.000,E1 271.892} C_DIS
LIN {X -0.052,Y -473.480,Z 999.508,A 0.000,B 0.000,C 90.000,E1 271.375} C_DIS
LIN {X 0.146,Y -468.106,Z 999.505,A 0.000,B 0.000,C 90.000,E1 270.859} C_DIS
LIN {X 0.195,Y -462.061,Z 999.502,A 0.000,B 0.000,C 90.000,E1 270.401} C_DIS
LIN {X -0.197,Y -455.547,Z 999.500,A 0.000,B 0.000,C 90.000,E1 270.057} C_DIS
LIN {X -0.110,Y -448.667,Z 999.498,A 0.000,B 0.000,C 90.000,E1 269.714} C_DIS
LIN {X -0.013,Y -441.527,Z 999.497,A 0.000,B 0.000,C 90.000,E1 269.427} C_DIS
LIN {X 0.057,Y -434.038,Z 999.496,A 0.000,B 0.000,C 90.000,E1 269.198} C_DIS
LIN {X 0.075,Y -425.826,Z 999.495,A 0.000,B 0.000,C 90.000,E1 269.026} C_DIS
LIN {X 0.008,Y -417.227,Z 999.494,A 0.000,B 0.000,C 90.000,E1 268.912} C_DIS
LIN {X 0.011,Y -405.202,Z 999.493,A 0.000,B 0.000,C 90.000,E1 268.797} C_DIS
LIN {X -0.133,Y -399.700,Z 999.493,A 0.000,B 0.000,C 90.000,E1 268.797} C_DIS
LIN {X -0.081,Y -181.269,Z 999.493,A 0.000,B 0.000,C 90.000,E1 268.797} C_DIS
LIN {X -0.002,Y -180.906,Z 999.474,A 0.000,B 0.000,C 90.000,E1 265.355} C_DIS
LIN {X 0.072,Y -180.681,Z 999.469,A 0.000,B 0.000,C 90.000,E1 264.489} C_DIS
LIN {X -0.030,Y -178.764,Z 999.441,A 0.000,B 0.000,C 90.000,E1 259.454} C_DIS
LIN {X 0.042,Y -175.811,Z 999.413,A 0.000,B 0.000,C 90.000,E1 254.338} C_DIS
LIN {X 0.037,Y -171.997,Z 999.385,A 0.000,B 0.000,C 90.000,E1 249.209} C_DIS
LIN {X 0.011,Y -171.411,Z 999.380,A 0.000,B 0.000,C 90.000,E1 248.358} C_DIS
LIN {X 0.058,Y -167.651,Z 999.356,A 0.000,B 0.000,C 90.000,E1 244.024} C_DIS
LIN {X 0.073,Y -166.315,Z 999.346,A 0.000,B 0.000,C 90.000,E1 242.281} C_DIS
LIN {X 0.067,Y -163.057,Z 999.327,A 0.000,B 0.000,C 90.000,E1 238.791} C_DIS
LIN {X 0.028,Y -160.992,Z 999.312,A 0.000,B 0.000,C 90.000,E1 236.167} C_DIS
LIN {X 0.006,Y -157.740,Z 999.292,A 0.000,B 0.000,C 90.000,E1 232.637} C_DIS
LIN {X -0.057,Y -155.779,Z 999.278,A 0.000,B 0.000,C 90.000,E1 229.989} C_DIS
LIN {X -0.001,Y -152.033,Z 999.253,A 0.000,B 0.000,C 90.000,E1 225.486} C_DIS
LIN {X 0.016,Y -150.281,Z 999.238,A 0.000,B 0.000,C 90.000,E1 222.771} C_DIS
LIN {X -0.057,Y -147.031,Z 999.212,A 0.000,B 0.000,C 90.000,E1 218.257} C_DIS
LIN {X -0.064,Y -145.612,Z 999.197,A 0.000,B 0.000,C 90.000,E1 215.518} C_DIS
LIN {X -0.065,Y -142.997,Z 999.172,A 0.000,B 0.000,C 90.000,E1 210.924} C_DIS
LIN {X -0.007,Y -141.624,Z 999.151,A 0.000,B 0.000,C 90.000,E1 207.206} C_DIS
LIN {X -0.082,Y -139.432,Z 999.115,A 0.000,B 0.000,C 90.000,E1 200.737} C_DIS
LIN {X -0.027,Y -139.163,Z 999.105,A 0.000,B 0.000,C 90.000,E1 198.852} C_DIS
LIN {X 0.010,Y -138.340,Z 999.058,A 0.000,B 0.000,C 90.000,E1 190.433} C_DIS
LIN {X 0.017,Y -139.477,Z 999.006,A 0.000,B 0.000,C 90.000,E1 181.088} C_DIS
LIN {X -0.042,Y -141.062,Z 998.975,A 0.000,B 0.000,C 90.000,E1 175.527} C_DIS
LIN {X 0.053,Y -142.435,Z 998.960,A 0.000,B 0.000,C 90.000,E1 172.704} C_DIS
LIN {X -0.028,Y -144.674,Z 998.934,A 0.000,B 0.000,C 90.000,E1 168.117} C_DIS
LIN {X -0.045,Y -147.261,Z 998.914,A 0.000,B 0.000,C 90.000,E1 164.448} C_DIS
LIN {X -0.027,Y -150.579,Z 998.888,A 0.000,B 0.000,C 90.000,E1 159.880} C_DIS
LIN {X 0.051,Y -154.050,Z 998.868,A 0.000,B 0.000,C 90.000,E1 156.230} C_DIS
LIN {X -0.022,Y -157.467,Z 998.848,A 0.000,B 0.000,C 90.000,E1 152.666} C_DIS
LIN {X 0.066,Y -161.689,Z 998.828,A 0.000,B 0.000,C 90.000,E1 149.076} C_DIS
LIN {X -0.057,Y -165.883,Z 998.809,A 0.000,B 0.000,C 90.000,E1 145.595} C_DIS
LIN {X -0.067,Y -170.864,Z 998.789,A 0.000,B 0.000,C 90.000,E1 142.110} C_DIS
LIN {X -0.020,Y -175.733,Z 998.770,A 0.000,B 0.000,C 90.000,E1 138.647} C_DIS
LIN {X -0.031,Y -181.344,Z 998.751,A 0.000,B 0.000,C 90.000,E1 135.243} C_DIS
LIN {X 0.104,Y -186.833,Z 998.733,A 0.000,B 0.000,C 90.000,E1 131.838} C_DIS
LIN {X 0.058,Y -191.420,Z 998.719,A 0.000,B 0.000,C 90.000,E1 129.358} C_DIS
LIN {X 0.020,Y -196.073,Z 998.704,A 0.000,B 0.000,C 90.000,E1 126.710} C_DIS
LIN {X -0.020,Y -299.903,Z 998.704,A 0.000,B 0.000,C 90.000,E1 126.710} C_DIS
LIN {X -0.171,Y -305.188,Z 998.703,A 0.000,B 0.000,C 90.000,E1 126.583} C_DIS
LIN {X 0.106,Y -307.485,Z 998.702,A 0.000,B 0.000,C 90.000,E1 126.377} C_DIS
LIN {X -0.015,Y -310.590,Z 998.701,A 0.000,B 0.000,C 90.000,E1 126.091} C_DIS
LIN {X 0.050,Y -314.216,Z 998.697,A 0.000,B 0.000,C 90.000,E1 125.518} C_DIS
LIN {X 0.097,Y -315.686,Z 998.696,A 0.000,B 0.000,C 90.000,E1 125.185} C_DIS
LIN {X 0.080,Y -320.992,Z 998.687,A 0.000,B 0.000,C 90.000,E1 123.579} C_DIS
LIN {X 0.114,Y -331.243,Z 998.671,A 0.000,B 0.000,C 90.000,E1 120.718} C_DIS
LIN {X 0.058,Y -342.832,Z 998.655,A 0.000,B 0.000,C 90.000,E1 117.924} C_DIS
LIN {X -0.130,Y -355.857,Z 998.640,A 0.000,B 0.000,C 90.000,E1 115.207} C_DIS
LIN {X 0.156,Y -368.735,Z 998.627,A 0.000,B 0.000,C 90.000,E1 112.770} C_DIS
LIN {X 0.159,Y -382.931,Z 998.614,A 0.000,B 0.000,C 90.000,E1 110.429} C_DIS
LIN {X -0.122,Y -398.546,Z 998.601,A 0.000,B 0.000,C 90.000,E1 108.181} C_DIS
LIN {X 0.238,Y -415.690,Z 998.589,A 0.000,B 0.000,C 90.000,E1 105.898} C_DIS
LIN {X -0.121,Y -434.489,Z 998.576,A 0.000,B 0.000,C 90.000,E1 103.772} C_DIS
LIN {X -0.120,Y -454.481,Z 998.565,A 0.000,B 0.000,C 90.000,E1 101.715} C_DIS
LIN {X 0.083,Y -467.253,Z 998.558,A 0.000,B 0.000,C 90.000,E1 100.489} C_DIS
LIN {X 0.084,Y -469.325,Z 998.557,A 0.000,B 0.000,C 90.000,E1 100.254} C_DIS
LIN {X 0.084,Y -470.897,Z 998.556,A 0.000,B 0.000,C 90.000,E1 100.018} C_DIS
LIN {X -0.144,Y -472.181,Z 998.554,A 0.000,B 0.000,C 90.000,E1 99.792} C_DIS
LIN {X 0.175,Y -473.126,Z 998.553,A 0.000,B 0.000,C 90.000,E1 99.500} C_DIS
LIN {X -0.105,Y -474.174,Z 998.550,A 0.000,B 0.000,C 90.000,E1 99.029} C_DIS
LIN {X 0.011,Y -474.235,Z 998.547,A 0.000,B 0.000,C 90.000,E1 98.511} C_DIS
LIN {X 0.136,Y -473.322,Z 998.544,A 0.000,B 0.000,C 90.000,E1 97.992} C_DIS
LIN {X -0.204,Y -471.285,Z 998.542,A 0.000,B 0.000,C 90.000,E1 97.530} C_DIS
LIN {X -0.024,Y -467.968,Z 998.539,A 0.000,B 0.000,C 90.000,E1 97.004} C_DIS
LIN {X -0.023,Y -455.906,Z 998.529,A 0.000,B 0.000,C 90.000,E1 95.220} C_DIS
LIN {X -0.157,Y -438.435,Z 998.515,A 0.000,B 0.000,C 90.000,E1 92.636} C_DIS
LIN {X -0.207,Y -425.430,Z 998.503,A 0.000,B 0.000,C 90.000,E1 90.516} C_DIS
LIN {X 0.137,Y -409.089,Z 998.486,A 0.000,B 0.000,C 90.000,E1 87.478} C_DIS
LIN {X 0.158,Y -400.135,Z 998.477,A 0.000,B 0.000,C 90.000,E1 85.812} C_DIS
LIN {X 0.019,Y -390.978,Z 998.467,A 0.000,B 0.000,C 90.000,E1 84.147} C_DIS
LIN {X 0.184,Y -381.627,Z 998.458,A 0.000,B 0.000,C 90.000,E1 82.413} C_DIS
LIN {X 0.175,Y -372.008,Z 998.448,A 0.000,B 0.000,C 90.000,E1 80.679} C_DIS
LIN {X 0.135,Y -363.803,Z 998.440,A 0.000,B 0.000,C 90.000,E1 79.218} C_DIS
LIN {X -0.171,Y -350.429,Z 998.427,A 0.000,B 0.000,C 90.000,E1 76.881} C_DIS
LIN {X 0.120,Y -337.418,Z 998.413,A 0.000,B 0.000,C 90.000,E1 74.393} C_DIS
LIN {X 0.079,Y -321.877,Z 998.396,A 0.000,B 0.000,C 90.000,E1 71.275} C_DIS
LIN {X -0.087,Y -312.773,Z 998.385,A 0.000,B 0.000,C 90.000,E1 69.390} C_DIS
LIN {X 0.059,Y -299.323,Z 998.369,A 0.000,B 0.000,C 90.000,E1 66.433} C_DIS
LIN {X 0.060,Y -287.701,Z 998.354,A 0.000,B 0.000,C 90.000,E1 63.768} C_DIS
LIN {X 0.080,Y -277.691,Z 998.341,A 0.000,B 0.000,C 90.000,E1 61.385} C_DIS
LIN {X 0.068,Y -266.305,Z 998.326,A 0.000,B 0.000,C 90.000,E1 58.614} C_DIS
LIN {X -0.137,Y -253.973,Z 998.308,A 0.000,B 0.000,C 90.000,E1 55.468} C_DIS
LIN {X -0.097,Y -242.277,Z 998.290,A 0.000,B 0.000,C 90.000,E1 52.190} C_DIS
LIN {X -0.084,Y -232.380,Z 998.273,A 0.000,B 0.000,C 90.000,E1 49.218} C_DIS
LIN {X 0.131,Y -223.034,Z 998.256,A 0.000,B 0.000,C 90.000,E1 46.134} C_DIS
LIN {X 0.006,Y -213.127,Z 998.237,A 0.000,B 0.000,C 90.000,E1 42.690} C_DIS
LIN {X -0.065,Y -204.874,Z 998.220,A 0.000,B 0.000,C 90.000,E1 39.564} C_DIS
LIN {X -0.118,Y -197.268,Z 998.202,A 0.000,B 0.000,C 90.000,E1 36.377} C_DIS
LIN {X 0.002,Y -190.378,Z 998.184,A 0.000,B 0.000,C 90.000,E1 33.086} C_DIS
LIN {X -0.044,Y -184.328,Z 998.165,A 0.000,B 0.000,C 90.000,E1 29.795} C_DIS
LIN {X -0.020,Y -179.014,Z 998.147,A 0.000,B 0.000,C 90.000,E1 26.437} C_DIS
LIN {X 0.042,Y -174.490,Z 998.128,A 0.000,B 0.000,C 90.000,E1 23.025} C_DIS
LIN {X -0.053,Y -170.609,Z 998.109,A 0.000,B 0.000,C 90.000,E1 19.631} C_DIS
LIN {X -0.036,Y -166.835,Z 998.085,A 0.000,B 0.000,C 90.000,E1 15.300} C_DIS
LIN {X -0.070,Y -164.090,Z 998.061,A 0.000,B 0.000,C 90.000,E1 10.950} C_DIS
LIN {X 0.052,Y -161.997,Z 998.027,A 0.000,B 0.000,C 90.000,E1 4.759} C_DIS
LIN {X 0.074,Y -163.139,Z 997.963,A 0.000,B 0.000,C 90.000,E1 353.337} C_DIS
LIN {X -0.056,Y -165.864,Z 997.934,A 0.000,B 0.000,C 90.000,E1 348.117} C_DIS
LIN {X -0.003,Y -169.386,Z 997.910,A 0.000,B 0.000,C 90.000,E1 343.740} C_DIS
LIN {X -0.052,Y -173.007,Z 997.890,A 0.000,B 0.000,C 90.000,E1 340.296} C_DIS
LIN {X 0.007,Y -177.481,Z 997.871,A 0.000,B 0.000,C 90.000,E1 336.847} C_DIS
LIN {X -0.016,Y -182.732,Z 997.853,A 0.000,B 0.000,C 90.000,E1 333.461} C_DIS
LIN {X -0.078,Y -188.782,Z 997.834,A 0.000,B 0.000,C 90.000,E1 330.127} C_DIS
LIN {X 0.039,Y -195.509,Z 997.816,A 0.000,B 0.000,C 90.000,E1 326.786} C_DIS
LIN {X -0.002,Y -202.816,Z 997.797,A 0.000,B 0.000,C 90.000,E1 323.543} C_DIS
LIN {X 0.134,Y -211.689,Z 997.777,A 0.000,B 0.000,C 90.000,E1 319.908} C_DIS
LIN {X 0.004,Y -221.061,Z 997.758,A 0.000,B 0.000,C 90.000,E1 316.419} C_DIS
LIN {X -0.028,Y -231.173,Z 997.739,A 0.000,B 0.000,C 90.000,E1 312.975} C_DIS
LIN {X -0.023,Y -235.169,Z 997.732,A 0.000,B 0.000,C 90.000,E1 311.838} C_DIS
LIN {X -0.001,Y -241.183,Z 997.724,A 0.000,B 0.000,C 90.000,E1 310.334} C_DIS
LIN {X 0.104,Y -251.045,Z 997.712,A 0.000,B 0.000,C 90.000,E1 308.096} C_DIS
LIN {X -0.019,Y -263.991,Z 997.698,A 0.000,B 0.000,C 90.000,E1 305.598} C_DIS
LIN {X -0.173,Y -278.293,Z 997.684,A 0.000,B 0.000,C 90.000,E1 303.166} C_DIS
LIN {X 0.083,Y -293.545,Z 997.671,A 0.000,B 0.000,C 90.000,E1 300.718} C_DIS
LIN {X -0.095,Y -314.596,Z 997.654,A 0.000,B 0.000,C 90.000,E1 297.769} C_DIS
LIN {X 0.069,Y -330.155,Z 997.644,A 0.000,B 0.000,C 90.000,E1 295.848} C_DIS
LIN {X 0.156,Y -354.345,Z 997.629,A 0.000,B 0.000,C 90.000,E1 293.259} C_DIS
LIN {X 0.194,Y -373.405,Z 997.619,A 0.000,B 0.000,C 90.000,E1 291.408} C_DIS
LIN {X -0.129,Y -389.747,Z 997.611,A 0.000,B 0.000,C 90.000,E1 289.939} C_DIS
LIN {X -0.002,Y -403.127,Z 997.604,A 0.000,B 0.000,C 90.000,E1 288.671} C_DIS
LIN {X 0.106,Y -413.555,Z 997.598,A 0.000,B 0.000,C 90.000,E1 287.638} C_DIS
LIN {X 0.116,Y -421.052,Z 997.594,A 0.000,B 0.000,C 90.000,E1 286.858} C_DIS
LIN {X 0.073,Y -430.972,Z 997.588,A 0.000,B 0.000,C 90.000,E1 285.788} C_DIS
LIN {X 0.075,Y -440.260,Z 997.582,A 0.000,B 0.000,C 90.000,E1 284.717} C_DIS
LIN {X 0.186,Y -449.058,Z 997.576,A 0.000,B 0.000,C 90.000,E1 283.647} C_DIS
LIN {X -0.150,Y -457.218,Z 997.570,A 0.000,B 0.000,C 90.000,E1 282.647} C_DIS
LIN {X 0.052,Y -464.572,Z 997.564,A 0.000,B 0.000,C 90.000,E1 281.591} C_DIS
LIN {X -0.054,Y -469.658,Z 997.560,A 0.000,B 0.000,C 90.000,E1 280.838} C_DIS
LIN {X -0.034,Y -474.205,Z 997.556,A 0.000,B 0.000,C 90.000,E1 280.074} C_DIS
LIN {X -0.055,Y -478.191,Z 997.552,A 0.000,B 0.000,C 90.000,E1 279.321} C_DIS
LIN {X -0.042,Y -481.549,Z 997.548,A 0.000,B 0.000,C 90.000,E1 278.568} C_DIS
LIN {X 0.122,Y -483.419,Z 997.545,A 0.000,B 0.000,C 90.000,E1 278.049} C_DIS
LIN {X -0.185,Y -485.060,Z 997.542,A 0.000,B 0.000,C 90.000,E1 277.587} C_DIS
LIN {X -0.001,Y -486.448,Z 997.539,A 0.000,B 0.000,C 90.000,E1 277.068} C_DIS
LIN {X 0.195,Y -487.606,Z 997.536,A 0.000,B 0.000,C 90.000,E1 276.549} C_DIS
LIN {X -0.087,Y -488.522,Z 997.534,A 0.000,B 0.000,C 90.000,E1 276.087} C_DIS
LIN {X 0.124,Y -489.110,Z 997.531,A 0.000,B 0.000,C 90.000,E1 275.568} C_DIS
LIN {X -0.149,Y -489.367,Z 997.528,A 0.000,B 0.000,C 90.000,E1 275.106} C_DIS
LIN {X 0.067,Y -489.199,Z 997.526,A 0.000,B 0.000,C 90.000,E1 274.588} C_DIS
LIN {X -0.240,Y -488.544,Z 997.523,A 0.000,B 0.000,C 90.000,E1 274.131} C_DIS
LIN {X -0.026,Y -487.402,Z 997.520,A 0.000,B 0.000,C 90.000,E1 273.612} C_DIS
LIN {X 0.181,Y -485.681,Z 997.517,A 0.000,B 0.000,C 90.000,E1 273.094} C_DIS
LIN {X -0.130,Y -483.308,Z 997.515,A 0.000,B 0.000,C 90.000,E1 272.636} C_DIS
LIN {X 0.190,Y -481.861,Z 997.513,A 0.000,B 0.000,C 90.000,E1 272.350} C_DIS
LIN {X -0.138,Y -478.284,Z 997.510,A 0.000,B 0.000,C 90.000,E1 271.892} C_DIS
LIN {X 0.187,Y -476.198,Z 997.509,A 0.000,B 0.000,C 90.000,E1 271.604} C_DIS
LIN {X -0.164,Y -471.210,Z 997.506,A 0.000,B 0.000,C 90.000,E1 271.146} C_DIS
LIN {X 0.117,Y -465.399,Z 997.504,A 0.000,B 0.000,C 90.000,E1 270.630} C_DIS
LIN {X -0.073,Y -459.073,Z 997.501,A 0.000,B 0.000,C 90.000,E1 270.229} C_DIS
LIN {X -0.212,Y -452.466,Z 997.499,A 0.000,B 0.000,C 90.000,E1 269.885} C_DIS
LIN {X 0.067,Y -445.398,Z 997.497,A 0.000,B 0.000,C 90.000,E1 269.542} C_DIS
LIN {X -0.102,Y -438.017,Z 997.496,A 0.000,B 0.000,C 90.000,E1 269.312} C_DIS
LIN {X 0.122,Y -430.016,Z 997.495,A 0.000,B 0.000,C 90.000,E1 269.083} C_DIS
LIN {X -0.090,Y -421.665,Z 997.494,A 0.000,B 0.000,C 90.000,E1 268.969} C_DIS
LIN {X 0.077,Y -408.842,Z 997.493,A 0.000,B 0.000,C 90.000,E1 268.797} C_DIS
LIN {X 0.176,Y -400.177,Z 997.493,A 0.000,B 0.000,C 90.000,E1 268.740} C_DIS
LIN {X 0.058,Y -181.266,Z 997.493,A 0.000,B 0.000,C 90.000,E1 268.740} C_DIS
LIN {X -0.046,Y -180.906,Z 997.474,A 0.000,B 0.000,C 90.000,E1 265.355} C_DIS
LIN {X 0.027,Y -180.674,Z 997.469,A 0.000,B 0.000,C 90.000,E1 264.489} C_DIS
LIN {X -0.074,Y -178.756,Z 997.441,A 0.000,B 0.000,C 90.000,E1 259.454} C_DIS
LIN {X -0.002,Y -175.803,Z 997.413,A 0.000,B 0.000,C 90.000,E1 254.338} C_DIS
LIN {X -0.007,Y -171.989,Z 997.384,A 0.000,B 0.000,C 90.000,E1 249.209} C_DIS
LIN {X 0.031,Y -171.398,Z 997.380,A 0.000,B 0.000,C 90.000,E1 248.337} C_DIS
LIN {X 0.016,Y -167.640,Z 997.356,A 0.000,B 0.000,C 90.000,E1 244.024} C_DIS
LIN {X 0.031,Y -166.299,Z 997.346,A 0.000,B 0.000,C 90.000,E1 242.281} C_DIS
LIN {X 0.025,Y -163.045,Z 997.327,A 0.000,B 0.000,C 90.000,E1 238.791} C_DIS
LIN {X -0.013,Y -160.978,Z 997.312,A 0.000,B 0.000,C 90.000,E1 236.167} C_DIS
LIN {X -0.036,Y -157.728,Z 997.292,A 0.000,B 0.000,C 90.000,E1 232.637} C_DIS
LIN {X -0.097,Y -155.767,Z 997.278,A 0.000,B 0.000,C 90.000,E1 229.989} C_DIS
LIN {X -0.041,Y -152.022,Z 997.253,A 0.000,B 0.000,C 90.000,E1 225.486} C_DIS
LIN {X -0.024,Y -150.269,Z 997.238,A 0.000,B 0.000,C 90.000,E1 222.771} C_DIS
LIN {X -0.005,Y -147.022,Z 997.212,A 0.000,B 0.000,C 90.000,E1 218.222} C_DIS
LIN {X 0.015,Y -145.604,Z 997.197,A 0.000,B 0.000,C 90.000,E1 215.471} C_DIS
LIN {X 0.020,Y -142.990,Z 997.172,A 0.000,B 0.000,C 90.000,E1 210.875} C_DIS
LIN {X 0.019,Y -141.617,Z 997.151,A 0.000,B 0.000,C 90.000,E1 207.180} C_DIS
LIN {X 0.060,Y -139.430,Z 997.115,A 0.000,B 0.000,C 90.000,E1 200.663} C_DIS
LIN {X -0.021,Y -139.160,Z 997.105,A 0.000,B 0.000,C 90.000,E1 198.833} C_DIS
LIN {X -0.003,Y -138.342,Z 997.058,A 0.000,B 0.000,C 90.000,E1 190.423} C_DIS
LIN {X -0.021,Y -139.480,Z 997.006,A 0.000,B 0.000,C 90.000,E1 181.088} C_DIS
LIN {X 0.060,Y -141.069,Z 996.975,A 0.000,B 0.000,C 90.000,E1 175.469} C_DIS
LIN {X 0.014,Y -142.443,Z 996.959,A 0.000,B 0.000,C 90.000,E1 172.704} C_DIS
LIN {X -0.037,Y -144.683,Z 996.934,A 0.000,B 0.000,C 90.000,E1 168.105} C_DIS
LIN {X 0.057,Y -147.274,Z 996.913,A 0.000,B 0.000,C 90.000,E1 164.393} C_DIS
LIN {X -0.068,Y -150.592,Z 996.888,A 0.000,B 0.000,C 90.000,E1 159.880} C_DIS
LIN {X 0.010,Y -154.065,Z 996.868,A 0.000,B 0.000,C 90.000,E1 156.230} C_DIS
LIN {X 0.077,Y -157.483,Z 996.848,A 0.000,B 0.000,C 90.000,E1 152.615} C_DIS
LIN {X 0.024,Y -161.708,Z 996.828,A 0.000,B 0.000,C 90.000,E1 149.076} C_DIS
LIN {X 0.037,Y -165.902,Z 996.809,A 0.000,B 0.000,C 90.000,E1 145.548} C_DIS
LIN {X 0.024,Y -170.886,Z 996.789,A 0.000,B 0.000,C 90.000,E1 142.065} C_DIS
LIN {X 0.052,Y -175.755,Z 996.770,A 0.000,B 0.000,C 90.000,E1 138.609} C_DIS
LIN {X -0.075,Y -181.364,Z 996.751,A 0.000,B 0.000,C 90.000,E1 135.243} C_DIS
LIN {X 0.058,Y -186.857,Z 996.733,A 0.000,B 0.000,C 90.000,E1 131.838} C_DIS
LIN {X 0.012,Y -191.443,Z 996.719,A 0.000,B 0.000,C 90.000,E1 129.358} C_DIS
LIN {X 0.024,Y -196.006,Z 996.704,A 0.000,B 0.000,C 90.000,E1 126.744} C_DIS
LIN {X 0.001,Y -299.575,Z 996.704,A 0.000,B 0.000,C 90.000,E1 126.744} C_DIS
LIN {X -0.091,Y -302.653,Z 996.704,A 0.000,B 0.000,C 90.000,E1 126.710} C_DIS
LIN {X 0.033,Y -307.961,Z 996.702,A 0.000,B 0.000,C 90.000,E1 126.377} C_DIS
LIN {X -0.089,Y -310.865,Z 996.700,A 0.000,B 0.000,C 90.000,E1 126.091} C_DIS
LIN {X -0.138,Y -312.890,Z 996.699,A 0.000,B 0.000,C 90.000,E1 125.804} C_DIS
LIN {X 0.069,Y -314.477,Z 996.697,A 0.000,B 0.000,C 90.000,E1 125.471} C_DIS
LIN {X 0.049,Y -315.857,Z 996.695,A 0.000,B 0.000,C 90.000,E1 125.152} C_DIS
LIN {X -0.156,Y -327.808,Z 996.676,A 0.000,B 0.000,C 90.000,E1 121.671} C_DIS
LIN {X 0.016,Y -338.957,Z 996.660,A 0.000,B 0.000,C 90.000,E1 118.821} C_DIS
LIN {X 0.028,Y -351.513,Z 996.645,A 0.000,B 0.000,C 90.000,E1 116.052} C_DIS
LIN {X 0.101,Y -365.581,Z 996.630,A 0.000,B 0.000,C 90.000,E1 113.334} C_DIS
LIN {X 0.160,Y -379.460,Z 996.617,A 0.000,B 0.000,C 90.000,E1 110.972} C_DIS
LIN {X -0.208,Y -394.732,Z 996.604,A 0.000,B 0.000,C 90.000,E1 108.725} C_DIS
LIN {X 0.051,Y -411.508,Z 996.591,A 0.000,B 0.000,C 90.000,E1 106.441} C_DIS
LIN {X 0.112,Y -429.907,Z 996.579,A 0.000,B 0.000,C 90.000,E1 104.245} C_DIS
LIN {X -0.080,Y -449.724,Z 996.568,A 0.000,B 0.000,C 90.000,E1 102.175} C_DIS
LIN {X -0.164,Y -467.527,Z 996.558,A 0.000,B 0.000,C 90.000,E1 100.489} C_DIS
LIN {X -0.176,Y -469.539,Z 996.557,A 0.000,B 0.000,C 90.000,E1 100.254} C_DIS
LIN {X -0.190,Y -471.067,Z 996.556,A 0.000,B 0.000,C 90.000,E1 100.018} C_DIS
LIN {X 0.127,Y -472.305,Z 996.554,A 0.000,B 0.000,C 90.000,E1 99.726} C_DIS
LIN {X -0.098,Y -473.213,Z 996.553,A 0.000,B 0.000,C 90.000,E1 99.500} C_DIS
LIN {X 0.089,Y -474.196,Z 996.550,A 0.000,B 0.000,C 90.000,E1 98.973} C_DIS
LIN {X 0.207,Y -474.198,Z 996.547,A 0.000,B 0.000,C 90.000,E1 98.454} C_DIS
LIN {X -0.136,Y -473.223,Z 996.544,A 0.000,B 0.000,C 90.000,E1 97.992} C_DIS
LIN {X 0.053,Y -471.105,Z 996.542,A 0.000,B 0.000,C 90.000,E1 97.466} C_DIS
LIN {X -0.195,Y -464.255,Z 996.536,A 0.000,B 0.000,C 90.000,E1 96.486} C_DIS
LIN {X -0.065,Y -453.943,Z 996.527,A 0.000,B 0.000,C 90.000,E1 94.935} C_DIS
LIN {X -0.080,Y -434.898,Z 996.511,A 0.000,B 0.000,C 90.000,E1 92.064} C_DIS
LIN {X -0.207,Y -422.225,Z 996.500,A 0.000,B 0.000,C 90.000,E1 89.943} C_DIS
LIN {X -0.116,Y -408.944,Z 996.486,A 0.000,B 0.000,C 90.000,E1 87.478} C_DIS
LIN {X -0.091,Y -399.988,Z 996.477,A 0.000,B 0.000,C 90.000,E1 85.812} C_DIS
LIN {X 0.161,Y -390.815,Z 996.467,A 0.000,B 0.000,C 90.000,E1 84.090} C_DIS
LIN {X -0.061,Y -381.448,Z 996.458,A 0.000,B 0.000,C 90.000,E1 82.413} C_DIS
LIN {X -0.066,Y -371.827,Z 996.448,A 0.000,B 0.000,C 90.000,E1 80.679} C_DIS
LIN {X -0.122,Y -361.945,Z 996.438,A 0.000,B 0.000,C 90.000,E1 78.926} C_DIS
LIN {X -0.042,Y -348.593,Z 996.425,A 0.000,B 0.000,C 90.000,E1 76.520} C_DIS
LIN {X 0.095,Y -334.043,Z 996.410,A 0.000,B 0.000,C 90.000,E1 73.740} C_DIS
LIN {X 0.110,Y -320.188,Z 996.394,A 0.000,B 0.000,C 90.000,E1 70.913} C_DIS
LIN {X -0.088,Y -311.083,Z 996.383,A 0.000,B 0.000,C 90.000,E1 69.028} C_DIS
LIN {X 0.121,Y -297.678,Z 996.367,A 0.000,B 0.000,C 90.000,E1 66.049} C_DIS
LIN {X 0.082,Y -286.082,Z 996.352,A 0.000,B 0.000,C 90.000,E1 63.384} C_DIS
LIN {X 0.069,Y -276.063,Z 996.339,A 0.000,B 0.000,C 90.000,E1 61.001} C_DIS
LIN {X -0.074,Y -264.707,Z 996.324,A 0.000,B 0.000,C 90.000,E1 58.250} C_DIS
LIN {X 0.015,Y -253.762,Z 996.308,A 0.000,B 0.000,C 90.000,E1 55.388} C_DIS
LIN {X 0.046,Y -242.059,Z 996.290,A 0.000,B 0.000,C 90.000,E1 52.110} C_DIS
LIN {X 0.050,Y -232.197,Z 996.273,A 0.000,B 0.000,C 90.000,E1 49.138} C_DIS
LIN {X -0.059,Y -222.829,Z 996.256,A 0.000,B 0.000,C 90.000,E1 46.134} C_DIS
LIN {X 0.120,Y -212.954,Z 996.237,A 0.000,B 0.000,C 90.000,E1 42.609} C_DIS
LIN {X 0.039,Y -204.717,Z 996.219,A 0.000,B 0.000,C 90.000,E1 39.483} C_DIS
LIN {X -0.023,Y -197.156,Z 996.202,A 0.000,B 0.000,C 90.000,E1 36.297} C_DIS
LIN {X -0.016,Y -190.300,Z 996.184,A 0.000,B 0.000,C 90.000,E1 33.038} C_DIS
LIN {X -0.057,Y -184.266,Z 996.165,A 0.000,B 0.000,C 90.000,E1 29.745} C_DIS
LIN {X 0.050,Y -178.965,Z 996.147,A 0.000,B 0.000,C 90.000,E1 26.360} C_DIS
LIN {X 0.105,Y -174.447,Z 996.128,A 0.000,B 0.000,C 90.000,E1 22.950} C_DIS
LIN {X -0.056,Y -170.581,Z 996.109,A 0.000,B 0.000,C 90.000,E1 19.577} C_DIS
LIN {X -0.036,Y -166.811,Z 996.085,A 0.000,B 0.000,C 90.000,E1 15.245} C_DIS
LIN {X -0.067,Y -164.099,Z 996.060,A 0.000,B 0.000,C 90.000,E1 10.894} C_DIS
LIN {X 0.002,Y -161.857,Z 996.021,A 0.000,B 0.000,C 90.000,E1 3.841} C_DIS
LIN {X 0.075,Y -163.172,Z 995.963,A 0.000,B 0.000,C 90.000,E1 353.337} C_DIS
LIN {X -0.055,Y -165.905,Z 995.934,A 0.000,B 0.000,C 90.000,E1 348.117} C_DIS
LIN {X 0.001,Y -169.438,Z 995.910,A 0.000,B 0.000,C 90.000,E1 343.740} C_DIS
LIN {X -0.047,Y -173.082,Z 995.890,A 0.000,B 0.000,C 90.000,E1 340.296} C_DIS
LIN {X 0.014,Y -177.551,Z 995.871,A 0.000,B 0.000,C 90.000,E1 336.847} C_DIS
LIN {X -0.007,Y -182.809,Z 995.853,A 0.000,B 0.000,C 90.000,E1 333.461} C_DIS
LIN {X -0.067,Y -188.864,Z 995.834,A 0.000,B 0.000,C 90.000,E1 330.127} C_DIS
LIN {X 0.053,Y -195.598,Z 995.816,A 0.000,B 0.000,C 90.000,E1 326.786} C_DIS
LIN {X 0.013,Y -202.910,Z 995.797,A 0.000,B 0.000,C 90.000,E1 323.543} C_DIS
LIN {X -0.009,Y -211.769,Z 995.778,A 0.000,B 0.000,C 90.000,E1 319.952} C_DIS
LIN {X 0.027,Y -221.134,Z 995.758,A 0.000,B 0.000,C 90.000,E1 316.419} C_DIS
LIN {X -0.003,Y -231.208,Z 995.739,A 0.000,B 0.000,C 90.000,E1 312.975} C_DIS
LIN {X 0.003,Y -235.207,Z 995.732,A 0.000,B 0.000,C 90.000,E1 311.838} C_DIS
LIN {X 0.008,Y -242.845,Z 995.722,A 0.000,B 0.000,C 90.000,E1 309.967} C_DIS
LIN {X 0.148,Y -252.913,Z 995.710,A 0.000,B 0.000,C 90.000,E1 307.729} C_DIS
LIN {X 0.061,Y -266.039,Z 995.696,A 0.000,B 0.000,C 90.000,E1 305.231} C_DIS
LIN {X -0.101,Y -282.654,Z 995.680,A 0.000,B 0.000,C 90.000,E1 302.467} C_DIS
LIN {X -0.047,Y -300.377,Z 995.665,A 0.000,B 0.000,C 90.000,E1 299.745} C_DIS
LIN {X 0.004,Y -317.136,Z 995.652,A 0.000,B 0.000,C 90.000,E1 297.436} C_DIS
LIN {X -0.044,Y -332.710,Z 995.642,A 0.000,B 0.000,C 90.000,E1 295.591} C_DIS
LIN {X -0.076,Y -359.755,Z 995.626,A 0.000,B 0.000,C 90.000,E1 292.770} C_DIS
LIN {X 0.057,Y -378.894,Z 995.616,A 0.000,B 0.000,C 90.000,E1 290.918} C_DIS
LIN {X 0.217,Y -392.521,Z 995.609,A 0.000,B 0.000,C 90.000,E1 289.631} C_DIS
LIN {X -0.024,Y -403.160,Z 995.604,A 0.000,B 0.000,C 90.000,E1 288.671} C_DIS
LIN {X 0.199,Y -413.375,Z 995.598,A 0.000,B 0.000,C 90.000,E1 287.638} C_DIS
LIN {X 0.166,Y -420.895,Z 995.594,A 0.000,B 0.000,C 90.000,E1 286.858} C_DIS
LIN {X 0.108,Y -430.821,Z 995.588,A 0.000,B 0.000,C 90.000,E1 285.788} C_DIS
LIN {X 0.110,Y -440.117,Z 995.582,A 0.000,B 0.000,C 90.000,E1 284.717} C_DIS
LIN {X 0.219,Y -448.923,Z 995.576,A 0.000,B 0.000,C 90.000,E1 283.647} C_DIS
LIN {X -0.118,Y -457.070,Z 995.570,A 0.000,B 0.000,C 90.000,E1 282.647} C_DIS
LIN {X 0.083,Y -464.425,Z 995.564,A 0.000,B 0.000,C 90.000,E1 281.591} C_DIS
LIN {X -0.179,Y -471.110,Z 995.559,A 0.000,B 0.000,C 90.000,E1 280.602} C_DIS
LIN {X -0.226,Y -475.543,Z 995.555,A 0.000,B 0.000,C 90.000,E1 279.849} C_DIS
LIN {X -0.160,Y -479.353,Z 995.550,A 0.000,B 0.000,C 90.000,E1 279.086} C_DIS
LIN {X -0.014,Y -481.558,Z 995.548,A 0.000,B 0.000,C 90.000,E1 278.568} C_DIS
LIN {X 0.150,Y -483.441,Z 995.545,A 0.000,B 0.000,C 90.000,E1 278.049} C_DIS
LIN {X -0.158,Y -485.111,Z 995.542,A 0.000,B 0.000,C 90.000,E1 277.587} C_DIS
LIN {X 0.027,Y -486.521,Z 995.539,A 0.000,B 0.000,C 90.000,E1 277.068} C_DIS
LIN {X -0.261,Y -487.688,Z 995.537,A 0.000,B 0.000,C 90.000,E1 276.606} C_DIS
LIN {X -0.058,Y -488.628,Z 995.534,A 0.000,B 0.000,C 90.000,E1 276.087} C_DIS
LIN {X 0.153,Y -489.216,Z 995.531,A 0.000,B 0.000,C 90.000,E1 275.568} C_DIS
LIN {X -0.118,Y -489.443,Z 995.528,A 0.000,B 0.000,C 90.000,E1 275.106} C_DIS
LIN {X 0.098,Y -489.289,Z 995.526,A 0.000,B 0.000,C 90.000,E1 274.588} C_DIS
LIN {X -0.209,Y -488.689,Z 995.523,A 0.000,B 0.000,C 90.000,E1 274.131} C_DIS
LIN {X 0.006,Y -487.565,Z 995.520,A 0.000,B 0.000,C 90.000,E1 273.612} C_DIS
LIN {X 0.213,Y -485.871,Z 995.517,A 0.000,B 0.000,C 90.000,E1 273.094} C_DIS
LIN {X -0.097,Y -483.528,Z 995.515,A 0.000,B 0.000,C 90.000,E1 272.636} C_DIS
LIN {X 0.063,Y -480.406,Z 995.512,A 0.000,B 0.000,C 90.000,E1 272.121} C_DIS
LIN {X 0.222,Y -476.467,Z 995.509,A 0.000,B 0.000,C 90.000,E1 271.604} C_DIS
LIN {X -0.129,Y -471.495,Z 995.506,A 0.000,B 0.000,C 90.000,E1 271.146} C_DIS
LIN {X 0.168,Y -465.735,Z 995.504,A 0.000,B 0.000,C 90.000,E1 270.630} C_DIS
LIN {X -0.041,Y -459.408,Z 995.501,A 0.000,B 0.000,C 90.000,E1 270.229} C_DIS
LIN {X -0.187,Y -452.837,Z 995.499,A 0.000,B 0.000,C 90.000,E1 269.885} C_DIS
LIN {X 0.101,Y -445.862,Z 995.497,A 0.000,B 0.000,C 90.000,E1 269.542} C_DIS
LIN {X -0.087,Y -438.523,Z 995.496,A 0.000,B 0.000,C 90.000,E1 269.312} C_DIS
LIN {X 0.089,Y -430.531,Z 995.495,A 0.000,B 0.000,C 90.000,E1 269.083} C_DIS
LIN {X -0.164,Y -421.914,Z 995.494,A 0.000,B 0.000,C 90.000,E1 268.969} C_DIS
LIN {X -0.004,Y -409.360,Z 995.493,A 0.000,B 0.000,C 90.000,E1 268.797} C_DIS
LIN {X 0.095,Y -401.143,Z 995.493,A 0.000,B 0.000,C 90.000,E1 268.740} C_DIS
LIN {X 0.021,Y -181.263,Z 995.493,A 0.000,B 0.000,C 90.000,E1 268.740} C_DIS
LIN {X -0.088,Y -180.905,Z 995.474,A 0.000,B 0.000,C 90.000,E1 265.355} C_DIS
LIN {X -0.014,Y -180.667,Z 995.469,A 0.000,B 0.000,C 90.000,E1 264.489} C_DIS
LIN {X 0.060,Y -178.748,Z 995.441,A 0.000,B 0.000,C 90.000,E1 259.398} C_DIS
LIN {X -0.042,Y -175.796,Z 995.413,A 0.000,B 0.000,C 90.000,E1 254.338} C_DIS
LIN {X -0.048,Y -171.981,Z 995.384,A 0.000,B 0.000,C 90.000,E1 249.209} C_DIS
LIN {X -0.009,Y -171.386,Z 995.380,A 0.000,B 0.000,C 90.000,E1 248.337} C_DIS
LIN {X -0.023,Y -167.630,Z 995.356,A 0.000,B 0.000,C 90.000,E1 244.024} C_DIS
LIN {X -0.009,Y -166.286,Z 995.346,A 0.000,B 0.000,C 90.000,E1 242.281} C_DIS
LIN {X -0.014,Y -163.034,Z 995.327,A 0.000,B 0.000,C 90.000,E1 238.791} C_DIS
LIN {X 0.038,Y -160.963,Z 995.312,A 0.000,B 0.000,C 90.000,E1 236.135} C_DIS
LIN {X -0.074,Y -157.716,Z 995.292,A 0.000,B 0.000,C 90.000,E1 232.637} C_DIS
LIN {X 0.085,Y -155.756,Z 995.277,A 0.000,B 0.000,C 90.000,E1 229.908} C_DIS
LIN {X -0.079,Y -152.012,Z 995.253,A 0.000,B 0.000,C 90.000,E1 225.486} C_DIS
LIN {X -0.060,Y -150.259,Z 995.237,A 0.000,B 0.000,C 90.000,E1 222.771} C_DIS
LIN {X 0.074,Y -147.013,Z 995.212,A 0.000,B 0.000,C 90.000,E1 218.177} C_DIS
LIN {X -0.021,Y -145.596,Z 995.197,A 0.000,B 0.000,C 90.000,E1 215.471} C_DIS
LIN {X -0.016,Y -142.983,Z 995.172,A 0.000,B 0.000,C 90.000,E1 210.875} C_DIS
LIN {X -0.016,Y -141.611,Z 995.151,A 0.000,B 0.000,C 90.000,E1 207.180} C_DIS
LIN {X 0.025,Y -139.427,Z 995.115,A 0.000,B 0.000,C 90.000,E1 200.663} C_DIS
LIN {X 0.076,Y -139.156,Z 995.104,A 0.000,B 0.000,C 90.000,E1 198.779} C_DIS
LIN {X -0.038,Y -138.343,Z 995.058,A 0.000,B 0.000,C 90.000,E1 190.423} C_DIS
LIN {X -0.057,Y -139.482,Z 995.006,A 0.000,B 0.000,C 90.000,E1 181.088} C_DIS
LIN {X 0.025,Y -141.075,Z 994.975,A 0.000,B 0.000,C 90.000,E1 175.469} C_DIS
LIN {X -0.022,Y -142.451,Z 994.959,A 0.000,B 0.000,C 90.000,E1 172.704} C_DIS
LIN {X 0.069,Y -144.692,Z 994.934,A 0.000,B 0.000,C 90.000,E1 168.049} C_DIS
LIN {X 0.021,Y -147.285,Z 994.913,A 0.000,B 0.000,C 90.000,E1 164.393} C_DIS
LIN {X 0.036,Y -150.604,Z 994.888,A 0.000,B 0.000,C 90.000,E1 159.826} C_DIS
LIN {X -0.028,Y -154.078,Z 994.868,A 0.000,B 0.000,C 90.000,E1 156.230} C_DIS
LIN {X 0.038,Y -157.498,Z 994.848,A 0.000,B 0.000,C 90.000,E1 152.615} C_DIS
LIN {X -0.016,Y -161.726,Z 994.828,A 0.000,B 0.000,C 90.000,E1 149.076} C_DIS
LIN {X -0.003,Y -165.920,Z 994.809,A 0.000,B 0.000,C 90.000,E1 145.548} C_DIS
LIN {X -0.016,Y -170.907,Z 994.789,A 0.000,B 0.000,C 90.000,E1 142.065} C_DIS
LIN {X 0.011,Y -175.775,Z 994.770,A 0.000,B 0.000,C 90.000,E1 138.609} C_DIS
LIN {X 0.012,Y -181.385,Z 994.751,A 0.000,B 0.000,C 90.000,E1 135.202} C_DIS
LIN {X 0.015,Y -186.881,Z 994.732,A 0.000,B 0.000,C 90.000,E1 131.838} C_DIS
LIN {X -0.032,Y -191.464,Z 994.719,A 0.000,B 0.000,C 90.000,E1 129.358} C_DIS
LIN {X -0.018,Y -195.943,Z 994.704,A 0.000,B 0.000,C 90.000,E1 126.790} C_DIS
LIN {X -0.079,Y -300.507,Z 994.704,A 0.000,B 0.000,C 90.000,E1 126.790} C_DIS
LIN {X 0.006,Y -302.019,Z 994.704,A 0.000,B 0.000,C 90.000,E1 126.744} C_DIS
LIN {X -0.050,Y -305.801,Z 994.703,A 0.000,B 0.000,C 90.000,E1 126.583} C_DIS
LIN {X 0.140,Y -308.026,Z 994.702,A 0.000,B 0.000,C 90.000,E1 126.377} C_DIS
LIN {X -0.158,Y -311.112,Z 994.700,A 0.000,B 0.000,C 90.000,E1 126.091} C_DIS
LIN {X -0.001,Y -313.100,Z 994.699,A 0.000,B 0.000,C 90.000,E1 125.758} C_DIS
LIN {X 0.086,Y -314.657,Z 994.697,A 0.000,B 0.000,C 90.000,E1 125.438} C_DIS
LIN {X 0.141,Y -315.969,Z 994.695,A 0.000,B 0.000,C 90.000,E1 125.105} C_DIS
LIN {X 0.127,Y -327.896,Z 994.676,A 0.000,B 0.000,C 90.000,E1 121.592} C_DIS
LIN {X -0.157,Y -339.059,Z 994.660,A 0.000,B 0.000,C 90.000,E1 118.821} C_DIS
LIN {X 0.006,Y -351.630,Z 994.645,A 0.000,B 0.000,C 90.000,E1 116.027} C_DIS
LIN {X -0.079,Y -365.714,Z 994.630,A 0.000,B 0.000,C 90.000,E1 113.334} C_DIS
LIN {X -0.023,Y -379.608,Z 994.617,A 0.000,B 0.000,C 90.000,E1 110.972} C_DIS
LIN {X -0.021,Y -394.898,Z 994.604,A 0.000,B 0.000,C 90.000,E1 108.671} C_DIS
LIN {X -0.140,Y -411.691,Z 994.591,A 0.000,B 0.000,C 90.000,E1 106.441} C_DIS
LIN {X -0.082,Y -430.110,Z 994.579,A 0.000,B 0.000,C 90.000,E1 104.245} C_DIS
LIN {X 0.171,Y -449.936,Z 994.567,A 0.000,B 0.000,C 90.000,E1 102.119} C_DIS
LIN {X 0.113,Y -467.716,Z 994.558,A 0.000,B 0.000,C 90.000,E1 100.433} C_DIS
LIN {X 0.090,Y -469.690,Z 994.557,A 0.000,B 0.000,C 90.000,E1 100.197} C_DIS
LIN {X 0.064,Y -471.190,Z 994.555,A 0.000,B 0.000,C 90.000,E1 99.962} C_DIS
LIN {X -0.082,Y -472.394,Z 994.554,A 0.000,B 0.000,C 90.000,E1 99.726} C_DIS
LIN {X 0.160,Y -473.273,Z 994.553,A 0.000,B 0.000,C 90.000,E1 99.443} C_DIS
LIN {X -0.119,Y -474.209,Z 994.550,A 0.000,B 0.000,C 90.000,E1 98.973} C_DIS
LIN {X -0.001,Y -474.167,Z 994.547,A 0.000,B 0.000,C 90.000,E1 98.454} C_DIS
LIN {X 0.125,Y -473.145,Z 994.544,A 0.000,B 0.000,C 90.000,E1 97.936} C_DIS
LIN {X -0.014,Y -472.221,Z 994.543,A 0.000,B 0.000,C 90.000,E1 97.701} C_DIS
LIN {X -0.154,Y -470.967,Z 994.541,A 0.000,B 0.000,C 90.000,E1 97.466} C_DIS
LIN {X 0.184,Y -457.304,Z 994.530,A 0.000,B 0.000,C 90.000,E1 95.391} C_DIS
LIN {X -0.066,Y -445.018,Z 994.520,A 0.000,B 0.000,C 90.000,E1 93.612} C_DIS
LIN {X -0.089,Y -428.289,Z 994.505,A 0.000,B 0.000,C 90.000,E1 90.974} C_DIS
LIN {X 0.014,Y -410.314,Z 994.487,A 0.000,B 0.000,C 90.000,E1 87.707} C_DIS
LIN {X 0.034,Y -401.397,Z 994.478,A 0.000,B 0.000,C 90.000,E1 86.045} C_DIS
LIN {X -0.049,Y -392.254,Z 994.469,A 0.000,B 0.000,C 90.000,E1 84.375} C_DIS
LIN {X 0.095,Y -382.892,Z 994.459,A 0.000,B 0.000,C 90.000,E1 82.648} C_DIS
LIN {X 0.166,Y -373.325,Z 994.450,A 0.000,B 0.000,C 90.000,E1 80.905} C_DIS
LIN {X 0.069,Y -363.475,Z 994.440,A 0.000,B 0.000,C 90.000,E1 79.162} C_DIS
LIN {X 0.096,Y -350.112,Z 994.427,A 0.000,B 0.000,C 90.000,E1 76.769} C_DIS
LIN {X 0.029,Y -335.496,Z 994.411,A 0.000,B 0.000,C 90.000,E1 74.031} C_DIS
LIN {X -0.014,Y -321.584,Z 994.396,A 0.000,B 0.000,C 90.000,E1 71.221} C_DIS
LIN {X -0.076,Y -312.466,Z 994.385,A 0.000,B 0.000,C 90.000,E1 69.316} C_DIS
LIN {X 0.070,Y -299.027,Z 994.369,A 0.000,B 0.000,C 90.000,E1 66.357} C_DIS
LIN {X 0.085,Y -288.804,Z 994.356,A 0.000,B 0.000,C 90.000,E1 64.024} C_DIS
LIN {X 0.133,Y -278.770,Z 994.343,A 0.000,B 0.000,C 90.000,E1 61.641} C_DIS
LIN {X 0.148,Y -267.354,Z 994.327,A 0.000,B 0.000,C 90.000,E1 58.869} C_DIS
LIN {X -0.064,Y -256.299,Z 994.312,A 0.000,B 0.000,C 90.000,E1 56.087} C_DIS
LIN {X -0.108,Y -244.411,Z 994.293,A 0.000,B 0.000,C 90.000,E1 52.844} C_DIS
LIN {X 0.138,Y -234.462,Z 994.277,A 0.000,B 0.000,C 90.000,E1 49.828} C_DIS
LIN {X 0.079,Y -224.979,Z 994.260,A 0.000,B 0.000,C 90.000,E1 46.824} C_DIS
LIN {X 0.002,Y -214.957,Z 994.241,A 0.000,B 0.000,C 90.000,E1 43.380} C_DIS
LIN {X -0.026,Y -206.605,Z 994.224,A 0.000,B 0.000,C 90.000,E1 40.253} C_DIS
LIN {X -0.071,Y -198.893,Z 994.206,A 0.000,B 0.000,C 90.000,E1 37.076} C_DIS
LIN {X 0.087,Y -191.888,Z 994.188,A 0.000,B 0.000,C 90.000,E1 33.785} C_DIS
LIN {X -0.080,Y -185.663,Z 994.170,A 0.000,B 0.000,C 90.000,E1 30.541} C_DIS
LIN {X -0.012,Y -180.189,Z 994.151,A 0.000,B 0.000,C 90.000,E1 27.180} C_DIS
LIN {X 0.072,Y -175.490,Z 994.132,A 0.000,B 0.000,C 90.000,E1 23.770} C_DIS
LIN {X 0.002,Y -171.467,Z 994.113,A 0.000,B 0.000,C 90.000,E1 20.375} C_DIS
LIN {X -0.060,Y -167.489,Z 994.089,A 0.000,B 0.000,C 90.000,E1 16.079} C_DIS
LIN {X -0.033,Y -164.568,Z 994.065,A 0.000,B 0.000,C 90.000,E1 11.715} C_DIS
LIN {X -0.021,Y -162.208,Z 994.031,A 0.000,B 0.000,C 90.000,E1 5.568} C_DIS
LIN {X 0.076,Y -163.208,Z 993.963,A 0.000,B 0.000,C 90.000,E1 353.337} C_DIS
LIN {X -0.052,Y -165.950,Z 993.934,A 0.000,B 0.000,C 90.000,E1 348.117} C_DIS
LIN {X -0.057,Y -168.699,Z 993.914,A 0.000,B 0.000,C 90.000,E1 344.629} C_DIS
LIN {X -0.012,Y -172.185,Z 993.895,A 0.000,B 0.000,C 90.000,E1 341.148} C_DIS
LIN {X -0.037,Y -176.444,Z 993.876,A 0.000,B 0.000,C 90.000,E1 337.720} C_DIS
LIN {X 0.081,Y -181.514,Z 993.857,A 0.000,B 0.000,C 90.000,E1 334.280} C_DIS
LIN {X 0.070,Y -187.389,Z 993.839,A 0.000,B 0.000,C 90.000,E1 330.923} C_DIS
LIN {X -0.110,Y -193.972,Z 993.820,A 0.000,B 0.000,C 90.000,E1 327.661} C_DIS
LIN {X 0.019,Y -201.126,Z 993.802,A 0.000,B 0.000,C 90.000,E1 324.356} C_DIS
LIN {X -0.088,Y -208.854,Z 993.784,A 0.000,B 0.000,C 90.000,E1 321.170} C_DIS
LIN {X 0.017,Y -218.044,Z 993.764,A 0.000,B 0.000,C 90.000,E1 317.595} C_DIS
LIN {X 0.061,Y -227.771,Z 993.745,A 0.000,B 0.000,C 90.000,E1 314.109} C_DIS
LIN {X -0.028,Y -232.543,Z 993.737,A 0.000,B 0.000,C 90.000,E1 312.609} C_DIS
LIN {X 0.115,Y -238.222,Z 993.728,A 0.000,B 0.000,C 90.000,E1 311.067} C_DIS
LIN {X -0.026,Y -251.257,Z 993.712,A 0.000,B 0.000,C 90.000,E1 308.141} C_DIS
LIN {X 0.103,Y -266.125,Z 993.696,A 0.000,B 0.000,C 90.000,E1 305.231} C_DIS
LIN {X -0.055,Y -282.703,Z 993.680,A 0.000,B 0.000,C 90.000,E1 302.467} C_DIS
LIN {X 0.003,Y -300.407,Z 993.665,A 0.000,B 0.000,C 90.000,E1 299.745} C_DIS
LIN {X -0.088,Y -317.158,Z 993.652,A 0.000,B 0.000,C 90.000,E1 297.462} C_DIS
LIN {X 0.110,Y -332.558,Z 993.642,A 0.000,B 0.000,C 90.000,E1 295.591} C_DIS
LIN {X -0.142,Y -359.401,Z 993.627,A 0.000,B 0.000,C 90.000,E1 292.823} C_DIS
LIN {X -0.096,Y -378.587,Z 993.616,A 0.000,B 0.000,C 90.000,E1 290.972} C_DIS
LIN {X 0.032,Y -392.233,Z 993.609,A 0.000,B 0.000,C 90.000,E1 289.685} C_DIS
LIN {X 0.110,Y -405.528,Z 993.602,A 0.000,B 0.000,C 90.000,E1 288.417} C_DIS
LIN {X -0.087,Y -413.174,Z 993.598,A 0.000,B 0.000,C 90.000,E1 287.692} C_DIS
LIN {X -0.160,Y -420.709,Z 993.594,A 0.000,B 0.000,C 90.000,E1 286.913} C_DIS
LIN {X -0.141,Y -430.494,Z 993.588,A 0.000,B 0.000,C 90.000,E1 285.843} C_DIS
LIN {X -0.150,Y -439.782,Z 993.582,A 0.000,B 0.000,C 90.000,E1 284.773} C_DIS
LIN {X -0.052,Y -448.624,Z 993.576,A 0.000,B 0.000,C 90.000,E1 283.703} C_DIS
LIN {X 0.047,Y -456.786,Z 993.570,A 0.000,B 0.000,C 90.000,E1 282.647} C_DIS
LIN {X 0.247,Y -464.143,Z 993.565,A 0.000,B 0.000,C 90.000,E1 281.591} C_DIS
LIN {X 0.138,Y -469.284,Z 993.560,A 0.000,B 0.000,C 90.000,E1 280.838} C_DIS
LIN {X -0.063,Y -475.395,Z 993.555,A 0.000,B 0.000,C 90.000,E1 279.849} C_DIS
LIN {X -0.073,Y -479.253,Z 993.550,A 0.000,B 0.000,C 90.000,E1 279.095} C_DIS
LIN {X 0.149,Y -481.465,Z 993.548,A 0.000,B 0.000,C 90.000,E1 278.568} C_DIS
LIN {X -0.166,Y -483.466,Z 993.545,A 0.000,B 0.000,C 90.000,E1 278.106} C_DIS
LIN {X 0.005,Y -485.128,Z 993.542,A 0.000,B 0.000,C 90.000,E1 277.587} C_DIS
LIN {X 0.190,Y -486.545,Z 993.539,A 0.000,B 0.000,C 90.000,E1 277.068} C_DIS
LIN {X -0.097,Y -487.739,Z 993.537,A 0.000,B 0.000,C 90.000,E1 276.606} C_DIS
LIN {X 0.107,Y -488.673,Z 993.534,A 0.000,B 0.000,C 90.000,E1 276.087} C_DIS
LIN {X -0.168,Y -489.314,Z 993.531,A 0.000,B 0.000,C 90.000,E1 275.625} C_DIS
LIN {X 0.047,Y -489.574,Z 993.528,A 0.000,B 0.000,C 90.000,E1 275.106} C_DIS
LIN {X -0.224,Y -489.440,Z 993.526,A 0.000,B 0.000,C 90.000,E1 274.645} C_DIS
LIN {X -0.043,Y -488.865,Z 993.523,A 0.000,B 0.000,C 90.000,E1 274.131} C_DIS
LIN {X 0.173,Y -487.763,Z 993.520,A 0.000,B 0.000,C 90.000,E1 273.612} C_DIS
LIN {X -0.131,Y -486.107,Z 993.517,A 0.000,B 0.000,C 90.000,E1 273.154} C_DIS
LIN {X 0.070,Y -483.802,Z 993.515,A 0.000,B 0.000,C 90.000,E1 272.636} C_DIS
LIN {X 0.231,Y -480.746,Z 993.512,A 0.000,B 0.000,C 90.000,E1 272.121} C_DIS
LIN {X -0.086,Y -476.852,Z 993.509,A 0.000,B 0.000,C 90.000,E1 271.661} C_DIS
LIN {X 0.214,Y -474.561,Z 993.508,A 0.000,B 0.000,C 90.000,E1 271.375} C_DIS
LIN {X 0.040,Y -471.976,Z 993.506,A 0.000,B 0.000,C 90.000,E1 271.146} C_DIS
LIN {X -0.167,Y -466.169,Z 993.504,A 0.000,B 0.000,C 90.000,E1 270.688} C_DIS
LIN {X -0.053,Y -463.241,Z 993.503,A 0.000,B 0.000,C 90.000,E1 270.458} C_DIS
LIN {X -0.032,Y -456.786,Z 993.500,A 0.000,B 0.000,C 90.000,E1 270.057} C_DIS
LIN {X 0.010,Y -450.048,Z 993.498,A 0.000,B 0.000,C 90.000,E1 269.714} C_DIS
LIN {X 0.029,Y -442.928,Z 993.497,A 0.000,B 0.000,C 90.000,E1 269.427} C_DIS
LIN {X -0.005,Y -435.427,Z 993.496,A 0.000,B 0.000,C 90.000,E1 269.198} C_DIS
LIN {X -0.062,Y -427.150,Z 993.495,A 0.000,B 0.000,C 90.000,E1 269.026} C_DIS
LIN {X -0.172,Y -418.854,Z 993.494,A 0.000,B 0.000,C 90.000,E1 268.912} C_DIS
LIN {X -0.058,Y -410.206,Z 993.493,A 0.000,B 0.000,C 90.000,E1 268.797} C_DIS
LIN {X -0.019,Y -400.699,Z 993.493,A 0.000,B 0.000,C 90.000,E1 268.740} C_DIS
LIN {X -0.032,Y -181.260,Z 993.493,A 0.000,B 0.000,C 90.000,E1 268.740} C_DIS
LIN {X 0.050,Y -180.905,Z 993.474,A 0.000,B 0.000,C 90.000,E1 265.298} C_DIS
LIN {X 0.000,Y -180.250,Z 993.465,A 0.000,B 0.000,C 90.000,E1 263.628} C_DIS
LIN {X 0.019,Y -178.741,Z 993.441,A 0.000,B 0.000,C 90.000,E1 259.398} C_DIS
LIN {X -0.084,Y -175.789,Z 993.413,A 0.000,B 0.000,C 90.000,E1 254.338} C_DIS
LIN {X -0.088,Y -171.973,Z 993.384,A 0.000,B 0.000,C 90.000,E1 249.209} C_DIS
LIN {X -0.050,Y -171.373,Z 993.380,A 0.000,B 0.000,C 90.000,E1 248.337} C_DIS
LIN {X -0.064,Y -167.620,Z 993.356,A 0.000,B 0.000,C 90.000,E1 244.024} C_DIS
LIN {X -0.048,Y -166.271,Z 993.346,A 0.000,B 0.000,C 90.000,E1 242.281} C_DIS
LIN {X -0.054,Y -163.023,Z 993.327,A 0.000,B 0.000,C 90.000,E1 238.791} C_DIS
LIN {X -0.002,Y -160.948,Z 993.312,A 0.000,B 0.000,C 90.000,E1 236.135} C_DIS
LIN {X -0.017,Y -157.705,Z 993.292,A 0.000,B 0.000,C 90.000,E1 232.603} C_DIS
LIN {X 0.046,Y -155.744,Z 993.277,A 0.000,B 0.000,C 90.000,E1 229.908} C_DIS
LIN {X -0.009,Y -152.002,Z 993.252,A 0.000,B 0.000,C 90.000,E1 225.445} C_DIS
LIN {X 0.004,Y -150.248,Z 993.237,A 0.000,B 0.000,C 90.000,E1 222.732} C_DIS
LIN {X 0.037,Y -147.005,Z 993.212,A 0.000,B 0.000,C 90.000,E1 218.177} C_DIS
LIN {X 0.026,Y -145.589,Z 993.197,A 0.000,B 0.000,C 90.000,E1 215.438} C_DIS
LIN {X -0.053,Y -142.977,Z 993.171,A 0.000,B 0.000,C 90.000,E1 210.875} C_DIS
LIN {X 0.073,Y -141.604,Z 993.151,A 0.000,B 0.000,C 90.000,E1 207.129} C_DIS
LIN {X -0.011,Y -139.424,Z 993.115,A 0.000,B 0.000,C 90.000,E1 200.663} C_DIS
LIN {X 0.040,Y -139.153,Z 993.104,A 0.000,B 0.000,C 90.000,E1 198.779} C_DIS
LIN {X 0.062,Y -138.344,Z 993.058,A 0.000,B 0.000,C 90.000,E1 190.366} C_DIS
LIN {X 0.048,Y -139.484,Z 993.006,A 0.000,B 0.000,C 90.000,E1 181.031} C_DIS
LIN {X -0.012,Y -141.081,Z 992.975,A 0.000,B 0.000,C 90.000,E1 175.469} C_DIS
LIN {X -0.058,Y -142.458,Z 992.959,A 0.000,B 0.000,C 90.000,E1 172.704} C_DIS
LIN {X 0.032,Y -144.701,Z 992.934,A 0.000,B 0.000,C 90.000,E1 168.049} C_DIS
LIN {X -0.017,Y -147.296,Z 992.913,A 0.000,B 0.000,C 90.000,E1 164.393} C_DIS
LIN {X -0.002,Y -150.616,Z 992.888,A 0.000,B 0.000,C 90.000,E1 159.826} C_DIS
LIN {X -0.065,Y -154.091,Z 992.868,A 0.000,B 0.000,C 90.000,E1 156.230} C_DIS
LIN {X 0.000,Y -157.513,Z 992.848,A 0.000,B 0.000,C 90.000,E1 152.615} C_DIS
LIN {X -0.056,Y -161.745,Z 992.828,A 0.000,B 0.000,C 90.000,E1 149.076} C_DIS
LIN {X 0.051,Y -165.937,Z 992.809,A 0.000,B 0.000,C 90.000,E1 145.515} C_DIS
LIN {X -0.057,Y -170.928,Z 992.789,A 0.000,B 0.000,C 90.000,E1 142.065} C_DIS
LIN {X -0.031,Y -175.796,Z 992.770,A 0.000,B 0.000,C 90.000,E1 138.609} C_DIS
LIN {X 0.097,Y -181.404,Z 992.751,A 0.000,B 0.000,C 90.000,E1 135.162} C_DIS
LIN {X -0.028,Y -186.904,Z 992.732,A 0.000,B 0.000,C 90.000,E1 131.838} C_DIS
LIN {X -0.076,Y -191.485,Z 992.719,A 0.000,B 0.000,C 90.000,E1 129.358} C_DIS
LIN {X 0.017,Y -195.860,Z 992.705,A 0.000,B 0.000,C 90.000,E1 126.824} C_DIS
LIN {X 0.153,Y -299.844,Z 992.705,A 0.000,B 0.000,C 90.000,E1 126.790} C_DIS
LIN {X 0.047,Y -301.270,Z 992.704,A 0.000,B 0.000,C 90.000,E1 126.790} C_DIS
LIN {X 0.148,Y -305.692,Z 992.703,A 0.000,B 0.000,C 90.000,E1 126.583} C_DIS
LIN {X 0.001,Y -308.090,Z 992.702,A 0.000,B 0.000,C 90.000,E1 126.423} C_DIS
LIN {X 0.206,Y -311.348,Z 992.700,A 0.000,B 0.000,C 90.000,E1 126.011} C_DIS
LIN {X 0.064,Y -313.297,Z 992.699,A 0.000,B 0.000,C 90.000,E1 125.724} C_DIS
LIN {X -0.080,Y -314.822,Z 992.697,A 0.000,B 0.000,C 90.000,E1 125.438} C_DIS
LIN {X 0.032,Y -317.094,Z 992.693,A 0.000,B 0.000,C 90.000,E1 124.771} C_DIS
LIN {X -0.042,Y -327.983,Z 992.675,A 0.000,B 0.000,C 90.000,E1 121.592} C_DIS
LIN {X 0.132,Y -339.160,Z 992.660,A 0.000,B 0.000,C 90.000,E1 118.743} C_DIS
LIN {X 0.148,Y -351.746,Z 992.644,A 0.000,B 0.000,C 90.000,E1 115.976} C_DIS
LIN {X 0.079,Y -365.846,Z 992.629,A 0.000,B 0.000,C 90.000,E1 113.281} C_DIS
LIN {X 0.150,Y -379.756,Z 992.616,A 0.000,B 0.000,C 90.000,E1 110.918} C_DIS
LIN {X -0.080,Y -395.062,Z 992.604,A 0.000,B 0.000,C 90.000,E1 108.652} C_DIS
LIN {X 0.066,Y -411.874,Z 992.591,A 0.000,B 0.000,C 90.000,E1 106.386} C_DIS
LIN {X 0.142,Y -430.313,Z 992.579,A 0.000,B 0.000,C 90.000,E1 104.189} C_DIS
LIN {X -0.017,Y -450.148,Z 992.567,A 0.000,B 0.000,C 90.000,E1 102.119} C_DIS
LIN {X -0.069,Y -467.900,Z 992.558,A 0.000,B 0.000,C 90.000,E1 100.433} C_DIS
LIN {X -0.109,Y -469.839,Z 992.557,A 0.000,B 0.000,C 90.000,E1 100.197} C_DIS
LIN {X -0.149,Y -471.312,Z 992.555,A 0.000,B 0.000,C 90.000,E1 99.962} C_DIS
LIN {X -0.054,Y -473.334,Z 992.552,A 0.000,B 0.000,C 90.000,E1 99.443} C_DIS
LIN {X 0.128,Y -474.223,Z 992.550,A 0.000,B 0.000,C 90.000,E1 98.916} C_DIS
LIN {X -0.221,Y -474.135,Z 992.547,A 0.000,B 0.000,C 90.000,E1 98.454} C_DIS
LIN {X -0.094,Y -473.062,Z 992.544,A 0.000,B 0.000,C 90.000,E1 97.936} C_DIS
LIN {X -0.232,Y -472.108,Z 992.543,A 0.000,B 0.000,C 90.000,E1 97.701} C_DIS
LIN {X 0.095,Y -470.818,Z 992.541,A 0.000,B 0.000,C 90.000,E1 97.409} C_DIS
LIN {X -0.031,Y -457.146,Z 992.530,A 0.000,B 0.000,C 90.000,E1 95.391} C_DIS
LIN {X -0.027,Y -446.628,Z 992.521,A 0.000,B 0.000,C 90.000,E1 93.841} C_DIS
LIN {X -0.011,Y -429.761,Z 992.507,A 0.000,B 0.000,C 90.000,E1 91.203} C_DIS
LIN {X -0.190,Y -410.206,Z 992.487,A 0.000,B 0.000,C 90.000,E1 87.707} C_DIS
LIN {X -0.167,Y -401.290,Z 992.478,A 0.000,B 0.000,C 90.000,E1 86.045} C_DIS
LIN {X 0.143,Y -392.143,Z 992.469,A 0.000,B 0.000,C 90.000,E1 84.318} C_DIS
LIN {X -0.100,Y -382.762,Z 992.459,A 0.000,B 0.000,C 90.000,E1 82.648} C_DIS
LIN {X -0.026,Y -373.200,Z 992.449,A 0.000,B 0.000,C 90.000,E1 80.905} C_DIS
LIN {X -0.121,Y -363.318,Z 992.440,A 0.000,B 0.000,C 90.000,E1 79.162} C_DIS
LIN {X -0.029,Y -351.630,Z 992.428,A 0.000,B 0.000,C 90.000,E1 77.061} C_DIS
LIN {X -0.145,Y -336.940,Z 992.413,A 0.000,B 0.000,C 90.000,E1 74.338} C_DIS
LIN {X -0.042,Y -322.993,Z 992.397,A 0.000,B 0.000,C 90.000,E1 71.511} C_DIS
LIN {X 0.041,Y -312.325,Z 992.385,A 0.000,B 0.000,C 90.000,E1 69.263} C_DIS
LIN {X 0.006,Y -300.351,Z 992.370,A 0.000,B 0.000,C 90.000,E1 66.666} C_DIS
LIN {X 0.058,Y -290.132,Z 992.357,A 0.000,B 0.000,C 90.000,E1 64.332} C_DIS
LIN {X 0.004,Y -280.061,Z 992.344,A 0.000,B 0.000,C 90.000,E1 61.975} C_DIS
LIN {X 0.054,Y -268.596,Z 992.329,A 0.000,B 0.000,C 90.000,E1 59.203} C_DIS
LIN {X -0.123,Y -257.497,Z 992.313,A 0.000,B 0.000,C 90.000,E1 56.421} C_DIS
LIN {X 0.074,Y -245.514,Z 992.295,A 0.000,B 0.000,C 90.000,E1 53.130} C_DIS
LIN {X -0.017,Y -234.304,Z 992.277,A 0.000,B 0.000,C 90.000,E1 49.828} C_DIS
LIN {X -0.073,Y -224.836,Z 992.260,A 0.000,B 0.000,C 90.000,E1 46.824} C_DIS
LIN {X 0.015,Y -214.826,Z 992.241,A 0.000,B 0.000,C 90.000,E1 43.338} C_DIS
LIN {X -0.034,Y -206.517,Z 992.223,A 0.000,B 0.000,C 90.000,E1 40.216} C_DIS
LIN {X -0.051,Y -198.824,Z 992.206,A 0.000,B 0.000,C 90.000,E1 37.030} C_DIS
LIN {X -0.049,Y -191.849,Z 992.188,A 0.000,B 0.000,C 90.000,E1 33.785} C_DIS
LIN {X 0.043,Y -185.635,Z 992.169,A 0.000,B 0.000,C 90.000,E1 30.463} C_DIS
LIN {X 0.020,Y -180.181,Z 992.151,A 0.000,B 0.000,C 90.000,E1 27.129} C_DIS
LIN {X -0.053,Y -175.481,Z 992.132,A 0.000,B 0.000,C 90.000,E1 23.770} C_DIS
LIN {X -0.061,Y -171.471,Z 992.113,A 0.000,B 0.000,C 90.000,E1 20.355} C_DIS
LIN {X -0.018,Y -167.505,Z 992.089,A 0.000,B 0.000,C 90.000,E1 16.024} C_DIS
LIN {X 0.012,Y -164.591,Z 992.065,A 0.000,B 0.000,C 90.000,E1 11.658} C_DIS
LIN {X 0.027,Y -162.242,Z 992.031,A 0.000,B 0.000,C 90.000,E1 5.511} C_DIS
LIN {X 0.078,Y -163.250,Z 991.963,A 0.000,B 0.000,C 90.000,E1 353.337} C_DIS
LIN {X -0.049,Y -166.003,Z 991.934,A 0.000,B 0.000,C 90.000,E1 348.117} C_DIS
LIN {X -0.052,Y -168.777,Z 991.914,A 0.000,B 0.000,C 90.000,E1 344.629} C_DIS
LIN {X -0.005,Y -172.272,Z 991.895,A 0.000,B 0.000,C 90.000,E1 341.148} C_DIS
LIN {X -0.028,Y -176.558,Z 991.876,A 0.000,B 0.000,C 90.000,E1 337.720} C_DIS
LIN {X 0.092,Y -181.625,Z 991.857,A 0.000,B 0.000,C 90.000,E1 334.280} C_DIS
LIN {X 0.084,Y -187.492,Z 991.839,A 0.000,B 0.000,C 90.000,E1 330.923} C_DIS
LIN {X -0.092,Y -194.078,Z 991.820,A 0.000,B 0.000,C 90.000,E1 327.661} C_DIS
LIN {X 0.040,Y -201.231,Z 991.802,A 0.000,B 0.000,C 90.000,E1 324.356} C_DIS
LIN {X -0.064,Y -208.946,Z 991.784,A 0.000,B 0.000,C 90.000,E1 321.170} C_DIS
LIN {X -0.103,Y -218.133,Z 991.764,A 0.000,B 0.000,C 90.000,E1 317.634} C_DIS
LIN {X 0.093,Y -227.858,Z 991.745,A 0.000,B 0.000,C 90.000,E1 314.109} C_DIS
LIN {X 0.006,Y -232.648,Z 991.737,A 0.000,B 0.000,C 90.000,E1 312.609} C_DIS
LIN {X 0.153,Y -238.342,Z 991.728,A 0.000,B 0.000,C 90.000,E1 311.067} C_DIS
LIN {X -0.142,Y -249.649,Z 991.714,A 0.000,B 0.000,C 90.000,E1 308.543} C_DIS
LIN {X 0.054,Y -262.349,Z 991.700,A 0.000,B 0.000,C 90.000,E1 305.964} C_DIS
LIN {X -0.039,Y -278.477,Z 991.684,A 0.000,B 0.000,C 90.000,E1 303.166} C_DIS
LIN {X 0.079,Y -293.650,Z 991.671,A 0.000,B 0.000,C 90.000,E1 300.747} C_DIS
LIN {X 0.064,Y -314.699,Z 991.654,A 0.000,B 0.000,C 90.000,E1 297.769} C_DIS
LIN {X -0.135,Y -327.410,Z 991.646,A 0.000,B 0.000,C 90.000,E1 296.232} C_DIS
LIN {X 0.038,Y -351.738,Z 991.631,A 0.000,B 0.000,C 90.000,E1 293.567} C_DIS
LIN {X -0.180,Y -370.895,Z 991.620,A 0.000,B 0.000,C 90.000,E1 291.716} C_DIS
LIN {X 0.195,Y -387.286,Z 991.612,A 0.000,B 0.000,C 90.000,E1 290.120} C_DIS
LIN {X -0.129,Y -400.708,Z 991.605,A 0.000,B 0.000,C 90.000,E1 288.906} C_DIS
LIN {X 0.158,Y -410.946,Z 991.599,A 0.000,B 0.000,C 90.000,E1 287.873} C_DIS
LIN {X -0.001,Y -420.917,Z 991.594,A 0.000,B 0.000,C 90.000,E1 286.858} C_DIS
LIN {X -0.088,Y -430.766,Z 991.588,A 0.000,B 0.000,C 90.000,E1 285.788} C_DIS
LIN {X -0.091,Y -440.050,Z 991.582,A 0.000,B 0.000,C 90.000,E1 284.717} C_DIS
LIN {X 0.014,Y -448.866,Z 991.576,A 0.000,B 0.000,C 90.000,E1 283.647} C_DIS
LIN {X 0.119,Y -456.971,Z 991.570,A 0.000,B 0.000,C 90.000,E1 282.591} C_DIS
LIN {X -0.131,Y -464.346,Z 991.564,A 0.000,B 0.000,C 90.000,E1 281.591} C_DIS
LIN {X 0.067,Y -471.063,Z 991.559,A 0.000,B 0.000,C 90.000,E1 280.546} C_DIS
LIN {X 0.024,Y -475.578,Z 991.554,A 0.000,B 0.000,C 90.000,E1 279.792} C_DIS
LIN {X 0.092,Y -479.445,Z 991.550,A 0.000,B 0.000,C 90.000,E1 279.029} C_DIS
LIN {X 0.241,Y -481.688,Z 991.547,A 0.000,B 0.000,C 90.000,E1 278.511} C_DIS
LIN {X -0.072,Y -483.664,Z 991.545,A 0.000,B 0.000,C 90.000,E1 278.049} C_DIS
LIN {X 0.101,Y -485.339,Z 991.542,A 0.000,B 0.000,C 90.000,E1 277.530} C_DIS
LIN {X -0.195,Y -486.740,Z 991.539,A 0.000,B 0.000,C 90.000,E1 277.068} C_DIS
LIN {X 0.003,Y -487.925,Z 991.536,A 0.000,B 0.000,C 90.000,E1 276.549} C_DIS
LIN {X 0.210,Y -488.832,Z 991.534,A 0.000,B 0.000,C 90.000,E1 276.030} C_DIS
LIN {X -0.065,Y -489.462,Z 991.531,A 0.000,B 0.000,C 90.000,E1 275.568} C_DIS
LIN {X 0.152,Y -489.699,Z 991.528,A 0.000,B 0.000,C 90.000,E1 275.049} C_DIS
LIN {X -0.118,Y -489.543,Z 991.525,A 0.000,B 0.000,C 90.000,E1 274.588} C_DIS
LIN {X 0.064,Y -488.911,Z 991.523,A 0.000,B 0.000,C 90.000,E1 274.073} C_DIS
LIN {X -0.206,Y -487.779,Z 991.520,A 0.000,B 0.000,C 90.000,E1 273.612} C_DIS
LIN {X 0.003,Y -486.074,Z 991.517,A 0.000,B 0.000,C 90.000,E1 273.094} C_DIS
LIN {X 0.177,Y -483.738,Z 991.514,A 0.000,B 0.000,C 90.000,E1 272.579} C_DIS
LIN {X -0.143,Y -480.633,Z 991.512,A 0.000,B 0.000,C 90.000,E1 272.121} C_DIS
LIN {X 0.020,Y -476.667,Z 991.509,A 0.000,B 0.000,C 90.000,E1 271.604} C_DIS
LIN {X 0.143,Y -471.713,Z 991.506,A 0.000,B 0.000,C 90.000,E1 271.088} C_DIS
LIN {X -0.056,Y -465.805,Z 991.503,A 0.000,B 0.000,C 90.000,E1 270.630} C_DIS
LIN {X 0.097,Y -462.927,Z 991.502,A 0.000,B 0.000,C 90.000,E1 270.401} C_DIS
LIN {X 0.177,Y -456.502,Z 991.500,A 0.000,B 0.000,C 90.000,E1 270.000} C_DIS
LIN {X -0.216,Y -449.788,Z 991.498,A 0.000,B 0.000,C 90.000,E1 269.714} C_DIS
LIN {X -0.182,Y -442.634,Z 991.497,A 0.000,B 0.000,C 90.000,E1 269.427} C_DIS
LIN {X -0.174,Y -435.116,Z 991.495,A 0.000,B 0.000,C 90.000,E1 269.198} C_DIS
LIN {X -0.201,Y -426.985,Z 991.494,A 0.000,B 0.000,C 90.000,E1 269.026} C_DIS
LIN {X 0.136,Y -414.444,Z 991.493,A 0.000,B 0.000,C 90.000,E1 268.797} C_DIS
LIN {X 0.059,Y -406.710,Z 991.493,A 0.000,B 0.000,C 90.000,E1 268.740} C_DIS
LIN {X -0.099,Y -401.764,Z 991.493,A 0.000,B 0.000,C 90.000,E1 268.740} C_DIS
LIN {X -0.067,Y -181.257,Z 991.493,A 0.000,B 0.000,C 90.000,E1 268.740} C_DIS
LIN {X 0.004,Y -180.903,Z 991.474,A 0.000,B 0.000,C 90.000,E1 265.298} C_DIS
LIN {X -0.046,Y -180.245,Z 991.465,A 0.000,B 0.000,C 90.000,E1 263.628} C_DIS
LIN {X -0.027,Y -178.732,Z 991.441,A 0.000,B 0.000,C 90.000,E1 259.398} C_DIS
LIN {X 0.040,Y -175.779,Z 991.413,A 0.000,B 0.000,C 90.000,E1 254.283} C_DIS
LIN {X 0.028,Y -171.964,Z 991.384,A 0.000,B 0.000,C 90.000,E1 249.156} C_DIS
LIN {X 0.066,Y -171.360,Z 991.379,A 0.000,B 0.000,C 90.000,E1 248.284} C_DIS
LIN {X 0.043,Y -167.609,Z 991.355,A 0.000,B 0.000,C 90.000,E1 243.973} C_DIS
LIN {X 0.054,Y -166.255,Z 991.346,A 0.000,B 0.000,C 90.000,E1 242.231} C_DIS
LIN {X 0.043,Y -163.010,Z 991.326,A 0.000,B 0.000,C 90.000,E1 238.742} C_DIS
LIN {X -0.045,Y -160.933,Z 991.312,A 0.000,B 0.000,C 90.000,E1 236.135} C_DIS
LIN {X 0.066,Y -157.693,Z 991.292,A 0.000,B 0.000,C 90.000,E1 232.557} C_DIS
LIN {X 0.004,Y -155.732,Z 991.277,A 0.000,B 0.000,C 90.000,E1 229.908} C_DIS
LIN {X 0.057,Y -151.990,Z 991.252,A 0.000,B 0.000,C 90.000,E1 225.405} C_DIS
LIN {X 0.073,Y -150.236,Z 991.237,A 0.000,B 0.000,C 90.000,E1 222.690} C_DIS
LIN {X -0.004,Y -146.996,Z 991.212,A 0.000,B 0.000,C 90.000,E1 218.177} C_DIS
LIN {X -0.014,Y -145.580,Z 991.197,A 0.000,B 0.000,C 90.000,E1 215.438} C_DIS
LIN {X -0.019,Y -142.969,Z 991.171,A 0.000,B 0.000,C 90.000,E1 210.846} C_DIS
LIN {X 0.034,Y -141.596,Z 991.151,A 0.000,B 0.000,C 90.000,E1 207.129} C_DIS
LIN {X -0.051,Y -139.421,Z 991.115,A 0.000,B 0.000,C 90.000,E1 200.663} C_DIS
LIN {X 0.000,Y -139.148,Z 991.104,A 0.000,B 0.000,C 90.000,E1 198.779} C_DIS
LIN {X 0.022,Y -138.345,Z 991.058,A 0.000,B 0.000,C 90.000,E1 190.366} C_DIS
LIN {X 0.008,Y -139.487,Z 991.006,A 0.000,B 0.000,C 90.000,E1 181.031} C_DIS
LIN {X -0.052,Y -141.088,Z 990.975,A 0.000,B 0.000,C 90.000,E1 175.469} C_DIS
LIN {X 0.043,Y -142.466,Z 990.959,A 0.000,B 0.000,C 90.000,E1 172.648} C_DIS
LIN {X -0.009,Y -144.710,Z 990.934,A 0.000,B 0.000,C 90.000,E1 168.049} C_DIS
LIN {X -0.058,Y -147.309,Z 990.913,A 0.000,B 0.000,C 90.000,E1 164.393} C_DIS
LIN {X -0.043,Y -150.630,Z 990.888,A 0.000,B 0.000,C 90.000,E1 159.826} C_DIS
LIN {X 0.033,Y -154.106,Z 990.868,A 0.000,B 0.000,C 90.000,E1 156.177} C_DIS
LIN {X -0.043,Y -157.530,Z 990.848,A 0.000,B 0.000,C 90.000,E1 152.615} C_DIS
LIN {X -0.099,Y -161.765,Z 990.828,A 0.000,B 0.000,C 90.000,E1 149.076} C_DIS
LIN {X 0.007,Y -165.958,Z 990.808,A 0.000,B 0.000,C 90.000,E1 145.515} C_DIS
LIN {X 0.003,Y -170.951,Z 990.789,A 0.000,B 0.000,C 90.000,E1 142.029} C_DIS
LIN {X 0.055,Y -175.820,Z 990.770,A 0.000,B 0.000,C 90.000,E1 138.566} C_DIS
LIN {X 0.051,Y -181.426,Z 990.751,A 0.000,B 0.000,C 90.000,E1 135.162} C_DIS
LIN {X -0.075,Y -186.930,Z 990.732,A 0.000,B 0.000,C 90.000,E1 131.838} C_DIS
LIN {X -0.003,Y -191.509,Z 990.718,A 0.000,B 0.000,C 90.000,E1 129.322} C_DIS
LIN {X -0.027,Y -195.799,Z 990.705,A 0.000,B 0.000,C 90.000,E1 126.870} C_DIS
LIN {X -0.093,Y -300.221,Z 990.705,A 0.000,B 0.000,C 90.000,E1 126.870} C_DIS
LIN {X -0.078,Y -304.174,Z 990.704,A 0.000,B 0.000,C 90.000,E1 126.744} C_DIS
LIN {X 0.061,Y -307.364,Z 990.703,A 0.000,B 0.000,C 90.000,E1 126.503} C_DIS
LIN {X 0.103,Y -311.050,Z 990.701,A 0.000,B 0.000,C 90.000,E1 126.091} C_DIS
LIN {X 0.016,Y -312.977,Z 990.699,A 0.000,B 0.000,C 90.000,E1 125.804} C_DIS
LIN {X -0.072,Y -314.493,Z 990.697,A 0.000,B 0.000,C 90.000,E1 125.518} C_DIS
LIN {X -0.017,Y -315.780,Z 990.695,A 0.000,B 0.000,C 90.000,E1 125.185} C_DIS
LIN {X -0.039,Y -327.669,Z 990.676,A 0.000,B 0.000,C 90.000,E1 121.671} C_DIS
LIN {X 0.133,Y -338.808,Z 990.660,A 0.000,B 0.000,C 90.000,E1 118.821} C_DIS
LIN {X -0.172,Y -351.353,Z 990.645,A 0.000,B 0.000,C 90.000,E1 116.104} C_DIS
LIN {X -0.118,Y -365.409,Z 990.630,A 0.000,B 0.000,C 90.000,E1 113.387} C_DIS
LIN {X -0.213,Y -379.276,Z 990.617,A 0.000,B 0.000,C 90.000,E1 111.046} C_DIS
LIN {X -0.092,Y -394.537,Z 990.604,A 0.000,B 0.000,C 90.000,E1 108.725} C_DIS
LIN {X 0.167,Y -411.300,Z 990.591,A 0.000,B 0.000,C 90.000,E1 106.441} C_DIS
LIN {X -0.188,Y -429.686,Z 990.579,A 0.000,B 0.000,C 90.000,E1 104.300} C_DIS
LIN {X -0.063,Y -449.494,Z 990.568,A 0.000,B 0.000,C 90.000,E1 102.187} C_DIS
LIN {X -0.058,Y -467.316,Z 990.558,A 0.000,B 0.000,C 90.000,E1 100.489} C_DIS
LIN {X -0.062,Y -469.368,Z 990.557,A 0.000,B 0.000,C 90.000,E1 100.254} C_DIS
LIN {X -0.066,Y -470.926,Z 990.556,A 0.000,B 0.000,C 90.000,E1 100.018} C_DIS
LIN {X 0.252,Y -472.193,Z 990.554,A 0.000,B 0.000,C 90.000,E1 99.726} C_DIS
LIN {X 0.026,Y -473.127,Z 990.553,A 0.000,B 0.000,C 90.000,E1 99.500} C_DIS
LIN {X 0.212,Y -474.154,Z 990.550,A 0.000,B 0.000,C 90.000,E1 98.973} C_DIS
LIN {X -0.139,Y -474.196,Z 990.547,A 0.000,B 0.000,C 90.000,E1 98.511} C_DIS
LIN {X -0.014,Y -473.264,Z 990.544,A 0.000,B 0.000,C 90.000,E1 97.992} C_DIS
LIN {X 0.114,Y -471.201,Z 990.542,A 0.000,B 0.000,C 90.000,E1 97.473} C_DIS
LIN {X 0.082,Y -466.143,Z 990.537,A 0.000,B 0.000,C 90.000,E1 96.720} C_DIS
LIN {X 0.057,Y -454.184,Z 990.527,A 0.000,B 0.000,C 90.000,E1 94.935} C_DIS
LIN {X -0.121,Y -436.849,Z 990.513,A 0.000,B 0.000,C 90.000,E1 92.350} C_DIS
LIN {X -0.204,Y -424.032,Z 990.501,A 0.000,B 0.000,C 90.000,E1 90.229} C_DIS
LIN {X 0.013,Y -409.180,Z 990.486,A 0.000,B 0.000,C 90.000,E1 87.478} C_DIS
LIN {X 0.040,Y -400.219,Z 990.477,A 0.000,B 0.000,C 90.000,E1 85.812} C_DIS
LIN {X -0.095,Y -391.030,Z 990.467,A 0.000,B 0.000,C 90.000,E1 84.147} C_DIS
LIN {X 0.072,Y -381.646,Z 990.458,A 0.000,B 0.000,C 90.000,E1 82.413} C_DIS
LIN {X 0.067,Y -372.039,Z 990.448,A 0.000,B 0.000,C 90.000,E1 80.679} C_DIS
LIN {X 0.011,Y -362.140,Z 990.438,A 0.000,B 0.000,C 90.000,E1 78.926} C_DIS
LIN {X 0.070,Y -350.452,Z 990.427,A 0.000,B 0.000,C 90.000,E1 76.825} C_DIS
LIN {X -0.093,Y -334.226,Z 990.410,A 0.000,B 0.000,C 90.000,E1 73.795} C_DIS
LIN {X -0.014,Y -321.891,Z 990.396,A 0.000,B 0.000,C 90.000,E1 71.275} C_DIS
LIN {X 0.042,Y -311.239,Z 990.384,A 0.000,B 0.000,C 90.000,E1 69.028} C_DIS
LIN {X -0.027,Y -299.284,Z 990.369,A 0.000,B 0.000,C 90.000,E1 66.433} C_DIS
LIN {X -0.008,Y -289.056,Z 990.356,A 0.000,B 0.000,C 90.000,E1 64.101} C_DIS
LIN {X 0.043,Y -278.983,Z 990.343,A 0.000,B 0.000,C 90.000,E1 61.719} C_DIS
LIN {X 0.062,Y -267.559,Z 990.328,A 0.000,B 0.000,C 90.000,E1 58.948} C_DIS
LIN {X -0.004,Y -256.474,Z 990.312,A 0.000,B 0.000,C 90.000,E1 56.135} C_DIS
LIN {X -0.038,Y -244.529,Z 990.294,A 0.000,B 0.000,C 90.000,E1 52.889} C_DIS
LIN {X 0.038,Y -233.389,Z 990.275,A 0.000,B 0.000,C 90.000,E1 49.542} C_DIS
LIN {X -0.047,Y -223.939,Z 990.258,A 0.000,B 0.000,C 90.000,E1 46.539} C_DIS
LIN {X -0.052,Y -215.095,Z 990.241,A 0.000,B 0.000,C 90.000,E1 43.461} C_DIS
LIN {X 0.060,Y -206.800,Z 990.224,A 0.000,B 0.000,C 90.000,E1 40.297} C_DIS
LIN {X -0.112,Y -199.099,Z 990.206,A 0.000,B 0.000,C 90.000,E1 37.156} C_DIS
LIN {X 0.055,Y -192.129,Z 990.188,A 0.000,B 0.000,C 90.000,E1 33.865} C_DIS
LIN {X -0.007,Y -185.878,Z 990.170,A 0.000,B 0.000,C 90.000,E1 30.590} C_DIS
LIN {X -0.024,Y -180.409,Z 990.151,A 0.000,B 0.000,C 90.000,E1 27.257} C_DIS
LIN {X -0.090,Y -175.677,Z 990.133,A 0.000,B 0.000,C 90.000,E1 23.898} C_DIS
LIN {X 0.070,Y -171.652,Z 990.114,A 0.000,B 0.000,C 90.000,E1 20.429} C_DIS
LIN {X 0.008,Y -167.654,Z 990.090,A 0.000,B 0.000,C 90.000,E1 16.134} C_DIS
LIN {X 0.037,Y -164.710,Z 990.065,A 0.000,B 0.000,C 90.000,E1 11.771} C_DIS
LIN {X 0.051,Y -162.314,Z 990.031,A 0.000,B 0.000,C 90.000,E1 5.625} C_DIS
LIN {X 0.080,Y -163.306,Z 989.963,A 0.000,B 0.000,C 90.000,E1 353.337} C_DIS
LIN {X -0.049,Y -165.512,Z 989.939,A 0.000,B 0.000,C 90.000,E1 348.993} C_DIS
LIN {X -0.047,Y -168.854,Z 989.914,A 0.000,B 0.000,C 90.000,E1 344.629} C_DIS
LIN {X 0.003,Y -172.382,Z 989.895,A 0.000,B 0.000,C 90.000,E1 341.148} C_DIS
LIN {X -0.017,Y -176.671,Z 989.876,A 0.000,B 0.000,C 90.000,E1 337.720} C_DIS
LIN {X -0.057,Y -181.743,Z 989.857,A 0.000,B 0.000,C 90.000,E1 334.332} C_DIS
LIN {X 0.102,Y -187.612,Z 989.839,A 0.000,B 0.000,C 90.000,E1 330.923} C_DIS
LIN {X -0.071,Y -194.194,Z 989.820,A 0.000,B 0.000,C 90.000,E1 327.661} C_DIS
LIN {X -0.099,Y -201.341,Z 989.802,A 0.000,B 0.000,C 90.000,E1 324.402} C_DIS
LIN {X -0.035,Y -209.047,Z 989.784,A 0.000,B 0.000,C 90.000,E1 321.170} C_DIS
LIN {X -0.076,Y -218.224,Z 989.765,A 0.000,B 0.000,C 90.000,E1 317.634} C_DIS
LIN {X 0.124,Y -227.978,Z 989.745,A 0.000,B 0.000,C 90.000,E1 314.109} C_DIS
LIN {X 0.038,Y -232.792,Z 989.737,A 0.000,B 0.000,C 90.000,E1 312.609} C_DIS
LIN {X 0.067,Y -237.006,Z 989.730,A 0.000,B 0.000,C 90.000,E1 311.472} C_DIS
LIN {X -0.105,Y -248.092,Z 989.716,A 0.000,B 0.000,C 90.000,E1 308.910} C_DIS
LIN {X -0.148,Y -260.554,Z 989.702,A 0.000,B 0.000,C 90.000,E1 306.377} C_DIS
LIN {X 0.079,Y -276.412,Z 989.686,A 0.000,B 0.000,C 90.000,E1 303.499} C_DIS
LIN {X -0.103,Y -291.513,Z 989.673,A 0.000,B 0.000,C 90.000,E1 301.131} C_DIS
LIN {X 0.081,Y -312.263,Z 989.656,A 0.000,B 0.000,C 90.000,E1 298.103} C_DIS
LIN {X -0.111,Y -324.890,Z 989.647,A 0.000,B 0.000,C 90.000,E1 296.539} C_DIS
LIN {X -0.066,Y -338.144,Z 989.639,A 0.000,B 0.000,C 90.000,E1 295.027} C_DIS
LIN {X 0.133,Y -362.749,Z 989.625,A 0.000,B 0.000,C 90.000,E1 292.461} C_DIS
LIN {X -0.091,Y -381.917,Z 989.615,A 0.000,B 0.000,C 90.000,E1 290.663} C_DIS
LIN {X -0.082,Y -395.434,Z 989.608,A 0.000,B 0.000,C 90.000,E1 289.396} C_DIS
LIN {X 0.037,Y -406.071,Z 989.602,A 0.000,B 0.000,C 90.000,E1 288.362} C_DIS
LIN {X 0.099,Y -413.750,Z 989.598,A 0.000,B 0.000,C 90.000,E1 287.583} C_DIS
LIN {X 0.100,Y -421.183,Z 989.593,A 0.000,B 0.000,C 90.000,E1 286.804} C_DIS
LIN {X -0.107,Y -428.522,Z 989.589,A 0.000,B 0.000,C 90.000,E1 286.024} C_DIS
LIN {X -0.139,Y -437.950,Z 989.583,A 0.000,B 0.000,C 90.000,E1 284.954} C_DIS
LIN {X -0.060,Y -446.874,Z 989.577,A 0.000,B 0.000,C 90.000,E1 283.883} C_DIS
LIN {X 0.019,Y -455.155,Z 989.571,A 0.000,B 0.000,C 90.000,E1 282.827} C_DIS
LIN {X 0.201,Y -462.669,Z 989.566,A 0.000,B 0.000,C 90.000,E1 281.771} C_DIS
LIN {X -0.074,Y -469.589,Z 989.560,A 0.000,B 0.000,C 90.000,E1 280.782} C_DIS
LIN {X -0.193,Y -475.721,Z 989.554,A 0.000,B 0.000,C 90.000,E1 279.782} C_DIS
LIN {X -0.206,Y -479.583,Z 989.550,A 0.000,B 0.000,C 90.000,E1 279.029} C_DIS
LIN {X -0.058,Y -481.854,Z 989.547,A 0.000,B 0.000,C 90.000,E1 278.511} C_DIS
LIN {X 0.108,Y -483.822,Z 989.544,A 0.000,B 0.000,C 90.000,E1 277.992} C_DIS
LIN {X -0.198,Y -485.513,Z 989.542,A 0.000,B 0.000,C 90.000,E1 277.530} C_DIS
LIN {X 0.049,Y -486.921,Z 989.539,A 0.000,B 0.000,C 90.000,E1 277.004} C_DIS
LIN {X 0.244,Y -488.068,Z 989.536,A 0.000,B 0.000,C 90.000,E1 276.486} C_DIS
LIN {X -0.089,Y -488.986,Z 989.533,A 0.000,B 0.000,C 90.000,E1 276.030} C_DIS
LIN {X 0.124,Y -489.604,Z 989.531,A 0.000,B 0.000,C 90.000,E1 275.511} C_DIS
LIN {X -0.146,Y -489.816,Z 989.528,A 0.000,B 0.000,C 90.000,E1 275.049} C_DIS
LIN {X 0.073,Y -489.607,Z 989.525,A 0.000,B 0.000,C 90.000,E1 274.531} C_DIS
LIN {X -0.196,Y -488.958,Z 989.522,A 0.000,B 0.000,C 90.000,E1 274.069} C_DIS
LIN {X -0.014,Y -487.801,Z 989.520,A 0.000,B 0.000,C 90.000,E1 273.555} C_DIS
LIN {X 0.195,Y -486.055,Z 989.517,A 0.000,B 0.000,C 90.000,E1 273.037} C_DIS
LIN {X -0.115,Y -483.708,Z 989.514,A 0.000,B 0.000,C 90.000,E1 272.579} C_DIS
LIN {X 0.048,Y -480.584,Z 989.511,A 0.000,B 0.000,C 90.000,E1 272.064} C_DIS
LIN {X 0.208,Y -476.562,Z 989.509,A 0.000,B 0.000,C 90.000,E1 271.547} C_DIS
LIN {X -0.142,Y -471.539,Z 989.506,A 0.000,B 0.000,C 90.000,E1 271.088} C_DIS
LIN {X 0.166,Y -465.623,Z 989.503,A 0.000,B 0.000,C 90.000,E1 270.573} C_DIS
LIN {X 0.022,Y -459.406,Z 989.501,A 0.000,B 0.000,C 90.000,E1 270.172} C_DIS
LIN {X -0.129,Y -452.768,Z 989.499,A 0.000,B 0.000,C 90.000,E1 269.828} C_DIS
LIN {X 0.130,Y -445.683,Z 989.497,A 0.000,B 0.000,C 90.000,E1 269.484} C_DIS
LIN {X -0.064,Y -438.266,Z 989.496,A 0.000,B 0.000,C 90.000,E1 269.255} C_DIS
LIN {X 0.162,Y -430.275,Z 989.495,A 0.000,B 0.000,C 90.000,E1 269.026} C_DIS
LIN {X -0.069,Y -422.181,Z 989.494,A 0.000,B 0.000,C 90.000,E1 268.912} C_DIS
LIN {X -0.030,Y -413.805,Z 989.493,A 0.000,B 0.000,C 90.000,E1 268.797} C_DIS
LIN {X -0.096,Y -405.871,Z 989.493,A 0.000,B 0.000,C 90.000,E1 268.740} C_DIS
LIN {X -0.174,Y -402.939,Z 989.493,A 0.000,B 0.000,C 90.000,E1 268.740} C_DIS
LIN {X 0.068,Y -181.254,Z 989.493,A 0.000,B 0.000,C 90.000,E1 268.682} C_DIS
LIN {X -0.058,Y -180.859,Z 989.472,A 0.000,B 0.000,C 90.000,E1 265.008} C_DIS
LIN {X -0.004,Y -178.972,Z 989.444,A 0.000,B 0.000,C 90.000,E1 259.926} C_DIS
LIN {X 0.006,Y -177.931,Z 989.435,A 0.000,B 0.000,C 90.000,E1 258.229} C_DIS
LIN {X 0.020,Y -175.570,Z 989.411,A 0.000,B 0.000,C 90.000,E1 253.976} C_DIS
LIN {X 0.027,Y -172.297,Z 989.387,A 0.000,B 0.000,C 90.000,E1 249.699} C_DIS
LIN {X 0.005,Y -171.776,Z 989.383,A 0.000,B 0.000,C 90.000,E1 248.847} C_DIS
LIN {X -0.022,Y -168.706,Z 989.363,A 0.000,B 0.000,C 90.000,E1 245.409} C_DIS
LIN {X 0.017,Y -166.770,Z 989.349,A 0.000,B 0.000,C 90.000,E1 242.794} C_DIS
LIN {X -0.064,Y -162.750,Z 989.325,A 0.000,B 0.000,C 90.000,E1 238.456} C_DIS
LIN {X -0.087,Y -161.440,Z 989.315,A 0.000,B 0.000,C 90.000,E1 236.707} C_DIS
LIN {X -0.045,Y -157.433,Z 989.290,A 0.000,B 0.000,C 90.000,E1 232.271} C_DIS
LIN {X -0.011,Y -155.439,Z 989.275,A 0.000,B 0.000,C 90.000,E1 229.585} C_DIS
LIN {X 0.038,Y -151.760,Z 989.251,A 0.000,B 0.000,C 90.000,E1 225.081} C_DIS
LIN {X 0.049,Y -149.961,Z 989.235,A 0.000,B 0.000,C 90.000,E1 222.366} C_DIS
LIN {X 0.077,Y -146.802,Z 989.210,A 0.000,B 0.000,C 90.000,E1 217.810} C_DIS
LIN {X -0.023,Y -145.379,Z 989.195,A 0.000,B 0.000,C 90.000,E1 215.105} C_DIS
LIN {X -0.031,Y -142.439,Z 989.164,A 0.000,B 0.000,C 90.000,E1 209.589} C_DIS
LIN {X 0.016,Y -141.431,Z 989.149,A 0.000,B 0.000,C 90.000,E1 206.796} C_DIS
LIN {X -0.003,Y -139.365,Z 989.113,A 0.000,B 0.000,C 90.000,E1 200.301} C_DIS
LIN {X -0.017,Y -138.811,Z 989.097,A 0.000,B 0.000,C 90.000,E1 197.511} C_DIS
LIN {X 0.033,Y -138.351,Z 989.056,A 0.000,B 0.000,C 90.000,E1 190.018} C_DIS
LIN {X 0.010,Y -139.541,Z 989.004,A 0.000,B 0.000,C 90.000,E1 180.688} C_DIS
LIN {X -0.037,Y -141.237,Z 988.973,A 0.000,B 0.000,C 90.000,E1 175.122} C_DIS
LIN {X 0.062,Y -142.608,Z 988.957,A 0.000,B 0.000,C 90.000,E1 172.299} C_DIS
LIN {X 0.015,Y -144.919,Z 988.932,A 0.000,B 0.000,C 90.000,E1 167.701} C_DIS
LIN {X 0.008,Y -147.547,Z 988.911,A 0.000,B 0.000,C 90.000,E1 164.031} C_DIS
LIN {X 0.040,Y -150.150,Z 988.891,A 0.000,B 0.000,C 90.000,E1 160.369} C_DIS
LIN {X 0.049,Y -153.519,Z 988.871,A 0.000,B 0.000,C 90.000,E1 156.741} C_DIS
LIN {X -0.029,Y -157.884,Z 988.846,A 0.000,B 0.000,C 90.000,E1 152.281} C_DIS
LIN {X -0.075,Y -162.172,Z 988.826,A 0.000,B 0.000,C 90.000,E1 148.742} C_DIS
LIN {X 0.039,Y -166.380,Z 988.807,A 0.000,B 0.000,C 90.000,E1 145.182} C_DIS
LIN {X 0.042,Y -171.396,Z 988.787,A 0.000,B 0.000,C 90.000,E1 141.698} C_DIS
LIN {X 0.081,Y -176.309,Z 988.768,A 0.000,B 0.000,C 90.000,E1 138.243} C_DIS
LIN {X -0.050,Y -180.596,Z 988.754,A 0.000,B 0.000,C 90.000,E1 135.729} C_DIS
LIN {X -0.073,Y -185.998,Z 988.735,A 0.000,B 0.000,C 90.000,E1 132.366} C_DIS
LIN {X -0.017,Y -190.632,Z 988.721,A 0.000,B 0.000,C 90.000,E1 129.850} C_DIS
LIN {X 0.096,Y -195.732,Z 988.705,A 0.000,B 0.000,C 90.000,E1 126.870} C_DIS
LIN {X 0.116,Y -299.772,Z 988.705,A 0.000,B 0.000,C 90.000,E1 126.870} C_DIS
LIN {X 0.034,Y -304.948,Z 988.704,A 0.000,B 0.000,C 90.000,E1 126.710} C_DIS
LIN {X -0.174,Y -307.232,Z 988.703,A 0.000,B 0.000,C 90.000,E1 126.583} C_DIS
LIN {X 0.162,Y -311.103,Z 988.701,A 0.000,B 0.000,C 90.000,E1 126.091} C_DIS
LIN {X 0.060,Y -313.004,Z 988.699,A 0.000,B 0.000,C 90.000,E1 125.804} C_DIS
LIN {X -0.043,Y -314.499,Z 988.697,A 0.000,B 0.000,C 90.000,E1 125.518} C_DIS
LIN {X -0.010,Y -316.782,Z 988.694,A 0.000,B 0.000,C 90.000,E1 124.865} C_DIS
LIN {X -0.010,Y -327.629,Z 988.676,A 0.000,B 0.000,C 90.000,E1 121.671} C_DIS
LIN {X 0.162,Y -338.765,Z 988.660,A 0.000,B 0.000,C 90.000,E1 118.821} C_DIS
LIN {X -0.142,Y -351.307,Z 988.645,A 0.000,B 0.000,C 90.000,E1 116.104} C_DIS
LIN {X -0.089,Y -365.361,Z 988.630,A 0.000,B 0.000,C 90.000,E1 113.387} C_DIS
LIN {X -0.185,Y -379.225,Z 988.617,A 0.000,B 0.000,C 90.000,E1 111.046} C_DIS
LIN {X -0.064,Y -394.483,Z 988.604,A 0.000,B 0.000,C 90.000,E1 108.725} C_DIS
LIN {X 0.196,Y -411.243,Z 988.591,A 0.000,B 0.000,C 90.000,E1 106.441} C_DIS
LIN {X -0.160,Y -429.625,Z 988.579,A 0.000,B 0.000,C 90.000,E1 104.300} C_DIS
LIN {X -0.036,Y -449.432,Z 988.568,A 0.000,B 0.000,C 90.000,E1 102.187} C_DIS
LIN {X -0.033,Y -467.257,Z 988.558,A 0.000,B 0.000,C 90.000,E1 100.489} C_DIS
LIN {X -0.034,Y -469.321,Z 988.557,A 0.000,B 0.000,C 90.000,E1 100.254} C_DIS
LIN {X -0.036,Y -470.887,Z 988.556,A 0.000,B 0.000,C 90.000,E1 100.018} C_DIS
LIN {X -0.184,Y -472.164,Z 988.554,A 0.000,B 0.000,C 90.000,E1 99.782} C_DIS
LIN {X 0.055,Y -473.104,Z 988.553,A 0.000,B 0.000,C 90.000,E1 99.500} C_DIS
LIN {X 0.242,Y -474.144,Z 988.550,A 0.000,B 0.000,C 90.000,E1 98.973} C_DIS
LIN {X -0.110,Y -474.198,Z 988.547,A 0.000,B 0.000,C 90.000,E1 98.511} C_DIS
LIN {X 0.016,Y -473.277,Z 988.544,A 0.000,B 0.000,C 90.000,E1 97.992} C_DIS
LIN {X 0.143,Y -471.230,Z 988.542,A 0.000,B 0.000,C 90.000,E1 97.473} C_DIS
LIN {X 0.110,Y -466.199,Z 988.537,A 0.000,B 0.000,C 90.000,E1 96.720} C_DIS
LIN {X 0.085,Y -454.240,Z 988.527,A 0.000,B 0.000,C 90.000,E1 94.935} C_DIS
LIN {X 0.173,Y -438.636,Z 988.514,A 0.000,B 0.000,C 90.000,E1 92.579} C_DIS
LIN {X 0.119,Y -425.647,Z 988.503,A 0.000,B 0.000,C 90.000,E1 90.458} C_DIS
LIN {X 0.047,Y -409.250,Z 988.486,A 0.000,B 0.000,C 90.000,E1 87.478} C_DIS
LIN {X 0.072,Y -400.279,Z 988.477,A 0.000,B 0.000,C 90.000,E1 85.812} C_DIS
LIN {X -0.011,Y -389.547,Z 988.466,A 0.000,B 0.000,C 90.000,E1 83.856} C_DIS
LIN {X 0.081,Y -380.111,Z 988.456,A 0.000,B 0.000,C 90.000,E1 82.129} C_DIS
LIN {X 0.101,Y -372.098,Z 988.448,A 0.000,B 0.000,C 90.000,E1 80.679} C_DIS
LIN {X 0.045,Y -362.180,Z 988.439,A 0.000,B 0.000,C 90.000,E1 78.926} C_DIS
LIN {X 0.103,Y -350.513,Z 988.427,A 0.000,B 0.000,C 90.000,E1 76.825} C_DIS
LIN {X -0.059,Y -334.290,Z 988.410,A 0.000,B 0.000,C 90.000,E1 73.795} C_DIS
LIN {X 0.020,Y -321.946,Z 988.396,A 0.000,B 0.000,C 90.000,E1 71.275} C_DIS
LIN {X -0.005,Y -309.770,Z 988.382,A 0.000,B 0.000,C 90.000,E1 68.720} C_DIS
LIN {X 0.013,Y -297.853,Z 988.367,A 0.000,B 0.000,C 90.000,E1 66.102} C_DIS
LIN {X 0.010,Y -287.625,Z 988.354,A 0.000,B 0.000,C 90.000,E1 63.768} C_DIS
LIN {X 0.029,Y -277.554,Z 988.341,A 0.000,B 0.000,C 90.000,E1 61.385} C_DIS
LIN {X 0.016,Y -266.159,Z 988.326,A 0.000,B 0.000,C 90.000,E1 58.614} C_DIS
LIN {X -0.047,Y -253.769,Z 988.308,A 0.000,B 0.000,C 90.000,E1 55.435} C_DIS
LIN {X 0.037,Y -241.958,Z 988.290,A 0.000,B 0.000,C 90.000,E1 52.145} C_DIS
LIN {X 0.030,Y -232.165,Z 988.273,A 0.000,B 0.000,C 90.000,E1 49.175} C_DIS
LIN {X -0.002,Y -221.660,Z 988.254,A 0.000,B 0.000,C 90.000,E1 45.769} C_DIS
LIN {X -0.056,Y -212.986,Z 988.237,A 0.000,B 0.000,C 90.000,E1 42.690} C_DIS
LIN {X 0.030,Y -204.823,Z 988.220,A 0.000,B 0.000,C 90.000,E1 39.519} C_DIS
LIN {X 0.097,Y -197.351,Z 988.202,A 0.000,B 0.000,C 90.000,E1 36.297} C_DIS
LIN {X -0.054,Y -190.561,Z 988.184,A 0.000,B 0.000,C 90.000,E1 33.086} C_DIS
LIN {X 0.067,Y -184.505,Z 988.165,A 0.000,B 0.000,C 90.000,E1 29.745} C_DIS
LIN {X 0.015,Y -179.227,Z 988.147,A 0.000,B 0.000,C 90.000,E1 26.411} C_DIS
LIN {X 0.004,Y -174.674,Z 988.128,A 0.000,B 0.000,C 90.000,E1 23.025} C_DIS
LIN {X 0.076,Y -170.841,Z 988.109,A 0.000,B 0.000,C 90.000,E1 19.577} C_DIS
LIN {X -0.061,Y -167.044,Z 988.085,A 0.000,B 0.000,C 90.000,E1 15.300} C_DIS
LIN {X 0.074,Y -164.330,Z 988.061,A 0.000,B 0.000,C 90.000,E1 10.894} C_DIS
LIN {X -0.011,Y -162.031,Z 988.022,A 0.000,B 0.000,C 90.000,E1 3.898} C_DIS
LIN {X 0.082,Y -163.367,Z 987.963,A 0.000,B 0.000,C 90.000,E1 353.337} C_DIS
LIN {X -0.045,Y -165.597,Z 987.939,A 0.000,B 0.000,C 90.000,E1 348.993} C_DIS
LIN {X -0.039,Y -168.946,Z 987.915,A 0.000,B 0.000,C 90.000,E1 344.629} C_DIS
LIN {X 0.013,Y -172.492,Z 987.895,A 0.000,B 0.000,C 90.000,E1 341.148} C_DIS
LIN {X -0.004,Y -176.798,Z 987.876,A 0.000,B 0.000,C 90.000,E1 337.720} C_DIS
LIN {X -0.040,Y -181.863,Z 987.857,A 0.000,B 0.000,C 90.000,E1 334.332} C_DIS
LIN {X 0.088,Y -186.187,Z 987.843,A 0.000,B 0.000,C 90.000,E1 331.769} C_DIS
LIN {X 0.048,Y -192.603,Z 987.825,A 0.000,B 0.000,C 90.000,E1 328.456} C_DIS
LIN {X 0.041,Y -199.626,Z 987.807,A 0.000,B 0.000,C 90.000,E1 325.182} C_DIS
LIN {X -0.061,Y -207.192,Z 987.789,A 0.000,B 0.000,C 90.000,E1 321.984} C_DIS
LIN {X 0.000,Y -216.206,Z 987.769,A 0.000,B 0.000,C 90.000,E1 318.405} C_DIS
LIN {X -0.095,Y -224.744,Z 987.752,A 0.000,B 0.000,C 90.000,E1 315.324} C_DIS
LIN {X 0.031,Y -230.465,Z 987.741,A 0.000,B 0.000,C 90.000,E1 313.380} C_DIS
LIN {X 0.147,Y -235.689,Z 987.733,A 0.000,B 0.000,C 90.000,E1 311.838} C_DIS
LIN {X -0.040,Y -244.924,Z 987.720,A 0.000,B 0.000,C 90.000,E1 309.644} C_DIS
